C09145=1192.403,-109.333,-39.221,179.092,5.592,149.257
C09146=1192.398,-109.084,-39.231,179.093,5.592,149.257
C09147=1192.393,-108.834,-39.240,179.096,5.592,149.256
C09148=1192.388,-108.584,-39.250,179.097,5.592,149.255
C09149=1192.382,-108.334,-39.259,179.100,5.592,149.255
C09150=1192.377,-108.085,-39.269,179.102,5.592,149.254
C09151=1192.372,-107.835,-39.278,179.104,5.593,149.254
C09152=1192.367,-107.585,-39.289,179.107,5.592,149.253
C09153=1192.361,-107.335,-39.298,179.109,5.593,149.252
C09154=1192.356,-107.085,-39.308,179.111,5.593,149.252
C09155=1192.351,-106.836,-39.317,179.113,5.593,149.251
C09156=1192.345,-106.586,-39.327,179.115,5.593,149.250
C09157=1192.340,-106.337,-39.337,179.118,5.593,149.250
C09158=1192.334,-106.087,-39.346,179.119,5.593,149.249
C09159=1192.330,-105.837,-39.356,179.122,5.594,149.249
C09160=1192.324,-105.586,-39.366,179.124,5.593,149.248
C09161=1192.319,-105.337,-39.376,179.126,5.594,149.247
C09162=1192.314,-105.088,-39.385,179.128,5.594,149.247
C09163=1192.308,-104.838,-39.395,179.131,5.594,149.246
C09164=1192.303,-104.588,-39.404,179.133,5.594,149.245
C09165=1192.298,-104.338,-39.415,179.135,5.595,149.245
C09166=1192.293,-104.088,-39.424,179.137,5.595,149.244
C09167=1192.287,-103.839,-39.434,179.140,5.595,149.244
C09168=1192.282,-103.589,-39.443,179.142,5.595,149.243
C09169=1192.276,-103.339,-39.453,179.144,5.595,149.242
C09170=1192.271,-103.090,-39.463,179.147,5.596,149.242
C09171=1192.266,-102.839,-39.473,179.148,5.596,149.241
C09172=1192.261,-102.590,-39.483,179.151,5.596,149.240
C09173=1192.256,-102.340,-39.493,179.153,5.596,149.240
C09174=1192.250,-102.090,-39.502,179.155,5.597,149.239
C09175=1192.245,-101.819,-39.513,179.157,5.596,149.239
C09176=1192.239,-101.547,-39.523,179.160,5.597,149.238
C09177=1192.233,-101.276,-39.534,179.163,5.597,149.237
C09178=1192.227,-101.005,-39.545,179.165,5.597,149.236
C09179=1192.222,-100.755,-39.555,179.167,5.597,149.236
C09180=1192.217,-100.505,-39.565,179.169,5.597,149.235
C09181=1192.212,-100.255,-39.575,179.172,5.597,149.234
C09182=1192.206,-100.005,-39.584,179.173,5.597,149.234
C09183=1192.201,-99.756,-39.594,179.176,5.598,149.233
C09184=1192.196,-99.506,-39.605,179.179,5.598,149.233
C09185=1192.190,-99.256,-39.615,179.180,5.598,149.232
C09186=1192.186,-99.007,-39.624,179.183,5.599,149.231
C09187=1192.180,-98.757,-39.634,179.185,5.598,149.231
C09188=1192.175,-98.506,-39.645,179.187,5.599,149.230
C09189=1192.170,-98.257,-39.654,179.189,5.599,149.229
C09190=1192.164,-98.008,-39.664,179.191,5.599,149.229
C09191=1192.158,-97.757,-39.674,179.193,5.599,149.228
C09192=1192.153,-97.508,-39.683,179.196,5.599,149.228
C09193=1192.148,-97.258,-39.694,179.198,5.599,149.227
C09194=1192.143,-97.008,-39.704,179.200,5.600,149.226
C09195=1192.138,-96.759,-39.714,179.203,5.600,149.226
C09196=1192.133,-96.509,-39.724,179.205,5.600,149.225
C09197=1192.127,-96.259,-39.734,179.207,5.601,149.224
C09198=1192.121,-96.009,-39.744,179.209,5.600,149.224
C09199=1192.117,-95.760,-39.754,179.212,5.601,149.223
C09200=1192.112,-95.510,-39.764,179.214,5.601,149.223
C09201=1192.106,-95.260,-39.775,179.216,5.601,149.222
C09202=1192.100,-95.011,-39.785,179.218,5.601,149.221
C09203=1192.096,-94.761,-39.794,179.221,5.601,149.221
C09204=1192.090,-94.511,-39.804,179.223,5.602,149.220
C09205=1192.085,-94.261,-39.814,179.225,5.602,149.219
C09206=1192.079,-94.011,-39.825,179.228,5.602,149.219
C09207=1192.075,-93.762,-39.835,179.229,5.602,149.218
C09208=1192.069,-93.512,-39.845,179.232,5.603,149.218
C09209=1192.064,-93.262,-39.855,179.234,5.602,149.217
C09210=1192.059,-93.012,-39.866,179.236,5.603,149.216
C09211=1192.054,-92.763,-39.875,179.238,5.603,149.216
C09212=1192.048,-92.513,-39.885,179.241,5.603,149.215
C09213=1192.043,-92.263,-39.896,179.243,5.604,149.214
C09214=1192.037,-92.014,-39.906,179.245,5.604,149.214
C09215=1192.032,-91.764,-39.916,179.248,5.604,149.213
C09216=1192.028,-91.514,-39.926,179.249,5.604,149.213
C09217=1192.022,-91.265,-39.937,179.252,5.604,149.212
C09218=1192.016,-91.015,-39.947,179.254,5.604,149.211
C09219=1192.011,-90.765,-39.957,179.256,5.605,149.211
C09220=1192.006,-90.515,-39.968,179.258,5.604,149.210
C09221=1192.000,-90.266,-39.978,179.261,5.605,149.209
C09222=1191.996,-90.016,-39.988,179.263,5.606,149.209
C09223=1191.990,-89.766,-39.998,179.265,5.605,149.208
C09224=1191.985,-89.517,-40.008,179.268,5.606,149.207
C09225=1191.980,-89.266,-40.019,179.270,5.606,149.207
C09226=1191.974,-89.017,-40.029,179.272,5.606,149.206
C09227=1191.969,-88.767,-40.039,179.274,5.606,149.205
C09228=1191.964,-88.517,-40.049,179.277,5.606,149.205
C09229=1191.959,-88.268,-40.059,179.279,5.607,149.204
C09230=1191.954,-88.018,-40.070,179.281,5.606,149.203
C09231=1191.948,-87.768,-40.080,179.284,5.607,149.203
C09232=1191.943,-87.519,-40.090,179.286,5.607,149.202
C09233=1191.938,-87.268,-40.101,179.288,5.607,149.202
C09234=1191.932,-87.019,-40.111,179.290,5.607,149.201
C09235=1191.927,-86.769,-40.122,179.293,5.608,149.200
C09236=1191.921,-86.519,-40.132,179.295,5.608,149.200
C09237=1191.917,-86.270,-40.142,179.297,5.608,149.199
C09238=1191.912,-86.020,-40.153,179.300,5.608,149.198
C09239=1191.906,-85.771,-40.163,179.302,5.608,149.198
C09240=1191.901,-85.520,-40.174,179.304,5.609,149.197
C09241=1191.896,-85.271,-40.184,179.307,5.609,149.197
C09242=1191.891,-85.021,-40.194,179.309,5.609,149.196
C09243=1191.885,-84.771,-40.205,179.311,5.609,149.195
C09244=1191.880,-84.522,-40.216,179.313,5.609,149.195
C09245=1191.875,-84.272,-40.226,179.316,5.610,149.194
C09246=1191.869,-84.022,-40.236,179.318,5.609,149.193
C09247=1191.864,-83.772,-40.247,179.320,5.610,149.193
C09248=1191.859,-83.523,-40.257,179.322,5.611,149.192
C09249=1191.854,-83.273,-40.268,179.325,5.610,149.191
C09250=1191.848,-83.023,-40.279,179.327,5.611,149.191
C09251=1191.843,-82.773,-40.289,179.329,5.611,149.190
C09252=1191.838,-82.524,-40.299,179.331,5.611,149.189
C09253=1191.832,-82.274,-40.310,179.334,5.611,149.189
C09254=1191.827,-82.024,-40.321,179.336,5.611,149.188
C09255=1191.822,-81.775,-40.331,179.338,5.612,149.188
C09256=1191.817,-81.525,-40.342,179.341,5.611,149.187
C09257=1191.811,-81.275,-40.352,179.343,5.612,149.186
C09258=1191.806,-81.025,-40.363,179.345,5.613,149.186
C09259=1191.801,-80.776,-40.373,179.347,5.612,149.185
C09260=1191.796,-80.526,-40.384,179.350,5.613,149.184
C09261=1191.790,-80.276,-40.394,179.352,5.613,149.184
C09262=1191.786,-80.027,-40.405,179.354,5.613,149.183
C09263=1191.780,-79.777,-40.416,179.357,5.614,149.182
C09264=1191.775,-79.527,-40.426,179.359,5.614,149.182
C09265=1191.770,-79.278,-40.437,179.361,5.614,149.181
C09266=1191.765,-79.028,-40.448,179.363,5.614,149.180
C09267=1191.759,-78.778,-40.458,179.366,5.614,149.180
C09268=1191.754,-78.528,-40.469,179.368,5.615,149.179
C09269=1191.749,-78.279,-40.479,179.370,5.614,149.179
C09270=1191.744,-78.029,-40.490,179.373,5.615,149.178
C09271=1191.739,-77.780,-40.501,179.375,5.615,149.177
C09272=1191.734,-77.529,-40.512,179.377,5.615,149.177
C09273=1191.728,-77.280,-40.522,179.380,5.616,149.176
C09274=1191.723,-77.030,-40.533,179.382,5.616,149.175
C09275=1191.717,-76.780,-40.544,179.384,5.616,149.175
C09276=1191.712,-76.530,-40.554,179.386,5.616,149.174
C09277=1191.707,-76.281,-40.565,179.389,5.617,149.174
C09278=1191.702,-76.031,-40.576,179.391,5.617,149.173
C09279=1191.696,-75.760,-40.588,179.393,5.617,149.172
C09280=1191.691,-75.490,-40.599,179.396,5.617,149.171
C09281=1191.685,-75.218,-40.611,179.399,5.617,149.171
C09282=1191.679,-74.947,-40.623,179.401,5.618,149.170
C09283=1191.673,-74.698,-40.633,179.403,5.618,149.169
C09284=1191.669,-74.448,-40.645,179.406,5.618,149.169
C09285=1191.663,-74.199,-40.655,179.408,5.619,149.168
C09286=1191.658,-73.949,-40.666,179.410,5.618,149.167
C09287=1191.653,-73.700,-40.676,179.412,5.619,149.167
C09288=1191.647,-73.450,-40.688,179.415,5.619,149.166
C09289=1191.642,-73.200,-40.699,179.417,5.619,149.166
C09290=1191.637,-72.950,-40.710,179.420,5.620,149.165
C09291=1191.632,-72.700,-40.720,179.422,5.620,149.164
C09292=1191.627,-72.451,-40.731,179.424,5.620,149.164
C09293=1191.621,-72.201,-40.743,179.427,5.620,149.163
C09294=1191.616,-71.952,-40.753,179.428,5.620,149.162
C09295=1191.611,-71.702,-40.764,179.431,5.621,149.162
C09296=1191.606,-71.452,-40.775,179.433,5.621,149.161
C09297=1191.600,-71.202,-40.786,179.436,5.621,149.160
C09298=1191.595,-70.952,-40.797,179.438,5.622,149.160
C09299=1191.589,-70.703,-40.808,179.440,5.621,149.159
C09300=1191.585,-70.453,-40.819,179.443,5.622,149.158
C09301=1191.580,-70.203,-40.829,179.445,5.623,149.158
C09302=1191.574,-69.954,-40.841,179.447,5.622,149.157
C09303=1191.569,-69.704,-40.852,179.450,5.623,149.157
C09304=1191.564,-69.454,-40.863,179.452,5.622,149.156
C09305=1191.559,-69.205,-40.874,179.454,5.623,149.155
C09306=1191.553,-68.954,-40.885,179.457,5.624,149.155
C09307=1191.548,-68.706,-40.896,179.459,5.623,149.154
C09308=1191.543,-68.456,-40.907,179.461,5.624,149.153
C09309=1191.538,-68.206,-40.918,179.464,5.624,149.153
C09310=1191.532,-67.956,-40.929,179.466,5.624,149.152
C09311=1191.527,-67.706,-40.940,179.468,5.624,149.151
C09312=1191.522,-67.457,-40.951,179.471,5.625,149.151
C09313=1191.516,-67.207,-40.963,179.473,5.625,149.150
C09314=1191.511,-66.957,-40.973,179.475,5.625,149.149
C09315=1191.507,-66.707,-40.984,179.478,5.626,149.149
C09316=1191.501,-66.458,-40.996,179.480,5.626,149.148
C09317=1191.496,-66.208,-41.007,179.482,5.626,149.148
C09318=1191.491,-65.958,-41.018,179.484,5.626,149.147
C09319=1191.486,-65.709,-41.029,179.487,5.626,149.146
C09320=1191.480,-65.459,-41.040,179.489,5.627,149.146
C09321=1191.475,-65.209,-41.051,179.491,5.627,149.145
C09322=1191.470,-64.960,-41.063,179.494,5.627,149.144
C09323=1191.464,-64.710,-41.074,179.496,5.628,149.144
C09324=1191.459,-64.460,-41.085,179.498,5.628,149.143
C09325=1191.454,-64.210,-41.097,179.501,5.628,149.142
C09326=1191.449,-63.961,-41.107,179.504,5.628,149.142
C09327=1191.444,-63.712,-41.119,179.505,5.628,149.141
C09328=1191.438,-63.461,-41.130,179.508,5.629,149.140
C09329=1191.433,-63.212,-41.141,179.510,5.629,149.140
C09330=1191.428,-62.963,-41.152,179.513,5.629,149.139
C09331=1191.423,-62.713,-41.164,179.515,5.630,149.139
C09332=1191.418,-62.462,-41.175,179.517,5.630,149.138
C09333=1191.412,-62.213,-41.186,179.519,5.630,149.137
C09334=1191.407,-61.964,-41.197,179.522,5.630,149.136
C09335=1191.402,-61.714,-41.209,179.524,5.631,149.136
C09336=1191.397,-61.464,-41.221,179.526,5.631,149.135
C09337=1191.391,-61.214,-41.231,179.529,5.631,149.135
C09338=1191.386,-60.964,-41.243,179.532,5.632,149.134
C09339=1191.381,-60.715,-41.254,179.533,5.632,149.133
C09340=1191.377,-60.465,-41.265,179.536,5.632,149.133
C09341=1191.371,-60.216,-41.277,179.539,5.632,149.132
C09342=1191.366,-59.966,-41.288,179.540,5.632,149.131
C09343=1191.360,-59.716,-41.299,179.543,5.633,149.131
C09344=1191.355,-59.466,-41.311,179.546,5.633,149.130
C09345=1191.350,-59.216,-41.322,179.548,5.633,149.129
C09346=1191.345,-58.967,-41.333,179.550,5.634,149.129
C09347=1191.339,-58.717,-41.345,179.553,5.634,149.128
C09348=1191.335,-58.468,-41.357,179.555,5.634,149.127
C09349=1191.329,-58.218,-41.368,179.557,5.634,149.127
C09350=1191.324,-57.969,-41.379,179.559,5.635,149.126
C09351=1191.319,-57.719,-41.391,179.562,5.635,149.126
C09352=1191.314,-57.469,-41.402,179.564,5.635,149.125
C09353=1191.309,-57.220,-41.414,179.567,5.636,149.124
C09354=1191.304,-56.970,-41.426,179.568,5.636,149.124
C09355=1191.299,-56.720,-41.436,179.571,5.636,149.123
C09356=1191.293,-56.470,-41.448,179.574,5.636,149.122
C09357=1191.288,-56.221,-41.459,179.576,5.637,149.122
C09358=1191.282,-55.971,-41.471,179.578,5.637,149.121
C09359=1191.277,-55.721,-41.483,179.581,5.637,149.120
C09360=1191.272,-55.471,-41.494,179.583,5.638,149.120
C09361=1191.266,-55.222,-41.506,179.585,5.637,149.119
C09362=1191.262,-54.972,-41.517,179.588,5.638,149.119
C09363=1191.256,-54.722,-41.529,179.590,5.639,149.118
C09364=1191.252,-54.473,-41.540,179.592,5.638,149.117
C09365=1191.246,-54.223,-41.552,179.595,5.639,149.116
C09366=1191.241,-53.973,-41.563,179.597,5.640,149.116
C09367=1191.236,-53.723,-41.575,179.599,5.639,149.115
C09368=1191.231,-53.475,-41.587,179.602,5.640,149.115
C09369=1191.226,-53.225,-41.599,179.605,5.640,149.114
C09370=1191.220,-52.975,-41.611,179.607,5.641,149.113
C09371=1191.215,-52.725,-41.622,179.609,5.641,149.113
C09372=1191.210,-52.476,-41.634,179.612,5.641,149.112
C09373=1191.205,-52.226,-41.645,179.614,5.641,149.111
C09374=1191.200,-51.976,-41.657,179.616,5.641,149.111
C09375=1191.194,-51.726,-41.669,179.619,5.642,149.110
C09376=1191.189,-51.477,-41.680,179.621,5.642,149.109
C09377=1191.184,-51.227,-41.692,179.623,5.642,149.109
C09378=1191.179,-50.978,-41.703,179.625,5.643,149.108
C09379=1191.174,-50.728,-41.715,179.628,5.643,149.107
C09380=1191.168,-50.478,-41.727,179.631,5.644,149.107
C09381=1191.164,-50.229,-41.739,179.633,5.643,149.106
C09382=1191.158,-49.979,-41.751,179.635,5.644,149.106
C09383=1191.152,-49.709,-41.763,179.638,5.645,149.105
C09384=1191.147,-49.439,-41.776,179.640,5.645,149.104
C09385=1191.142,-49.168,-41.788,179.643,5.645,149.104
C09386=1191.136,-48.898,-41.801,179.645,5.645,149.103
C09387=1191.131,-48.649,-41.814,179.648,5.645,149.102
C09388=1191.125,-48.399,-41.825,179.650,5.646,149.101
C09389=1191.120,-48.149,-41.837,179.653,5.646,149.101
C09390=1191.115,-47.899,-41.849,179.655,5.646,149.100
C09391=1191.110,-47.649,-41.861,179.657,5.647,149.100
C09392=1191.105,-47.400,-41.873,179.660,5.647,149.099
C09393=1191.100,-47.150,-41.884,179.662,5.647,149.098
C09394=1191.094,-46.900,-41.896,179.664,5.648,149.098
C09395=1191.089,-46.650,-41.908,179.667,5.648,149.097
C09396=1191.084,-46.401,-41.920,179.670,5.649,149.096
C09397=1191.079,-46.152,-41.932,179.672,5.648,149.096
C09398=1191.074,-45.902,-41.944,179.674,5.649,149.095
C09399=1191.068,-45.652,-41.956,179.677,5.650,149.094
C09400=1191.064,-45.403,-41.968,179.679,5.649,149.094
C09401=1191.058,-45.153,-41.980,179.681,5.650,149.093
C09402=1191.052,-44.904,-41.991,179.684,5.650,149.092
C09403=1191.047,-44.654,-42.004,179.686,5.651,149.092
C09404=1191.043,-44.405,-42.015,179.688,5.651,149.091
C09405=1191.037,-44.155,-42.027,179.691,5.651,149.090
C09406=1191.032,-43.905,-42.039,179.694,5.651,149.090
C09407=1191.027,-43.655,-42.052,179.696,5.652,149.089
C09408=1191.022,-43.406,-42.063,179.698,5.652,149.089
C09409=1191.017,-43.156,-42.075,179.700,5.652,149.088
C09410=1191.011,-42.906,-42.087,179.703,5.653,149.087
C09411=1191.006,-42.657,-42.099,179.705,5.654,149.087
C09412=1191.001,-42.407,-42.112,179.707,5.653,149.086
C09413=1190.995,-42.157,-42.124,179.710,5.654,149.085
C09414=1190.991,-41.908,-42.135,179.713,5.654,149.085
C09415=1190.986,-41.658,-42.148,179.714,5.654,149.084
C09416=1190.981,-41.408,-42.160,179.717,5.655,149.083
C09417=1190.976,-41.158,-42.172,179.720,5.655,149.083
C09418=1190.970,-40.908,-42.184,179.722,5.656,149.082
C09419=1190.965,-40.659,-42.196,179.724,5.655,149.081
C09420=1190.960,-40.410,-42.208,179.727,5.656,149.081
C09421=1190.955,-40.160,-42.220,179.729,5.656,149.080
C09422=1190.950,-39.910,-42.233,179.732,5.657,149.079
C09423=1190.944,-39.660,-42.245,179.734,5.657,149.079
C09424=1190.939,-39.411,-42.257,179.736,5.657,149.078
C09425=1190.934,-39.161,-42.269,179.739,5.658,149.078
C09426=1190.929,-38.912,-42.282,179.741,5.658,149.077
C09427=1190.923,-38.662,-42.294,179.744,5.658,149.076
C09428=1190.919,-38.413,-42.306,179.746,5.659,149.076
C09429=1190.913,-38.163,-42.317,179.748,5.659,149.075
C09430=1190.908,-37.914,-42.330,179.751,5.660,149.074
C09431=1190.903,-37.664,-42.342,179.753,5.659,149.074
C09432=1190.898,-37.414,-42.354,179.756,5.660,149.073
C09433=1190.893,-37.164,-42.367,179.758,5.661,149.072
C09434=1190.888,-36.914,-42.379,179.761,5.661,149.072
C09435=1190.882,-36.664,-42.391,179.763,5.661,149.071
C09436=1190.877,-36.415,-42.404,179.765,5.661,149.070
C09437=1190.872,-36.165,-42.416,179.768,5.662,149.070
C09438=1190.867,-35.916,-42.428,179.770,5.662,149.069
C09439=1190.862,-35.667,-42.441,179.773,5.663,149.068
C09440=1190.856,-35.417,-42.453,179.775,5.662,149.068
C09441=1190.851,-35.167,-42.465,179.777,5.663,149.067
C09442=1190.846,-34.917,-42.477,179.780,5.664,149.067
C09443=1190.841,-34.667,-42.490,179.782,5.664,149.066
C09444=1190.836,-34.418,-42.503,179.785,5.664,149.065
C09445=1190.830,-34.168,-42.515,179.787,5.664,149.064
C09446=1190.825,-33.919,-42.527,179.789,5.665,149.064
C09447=1190.820,-33.669,-42.539,179.792,5.666,149.063
C09448=1190.815,-33.419,-42.552,179.795,5.666,149.063
C09449=1190.810,-33.170,-42.564,179.797,5.666,149.062
C09450=1190.805,-32.920,-42.577,179.799,5.667,149.061
C09451=1190.800,-32.670,-42.589,179.802,5.667,149.061
C09452=1190.795,-32.421,-42.602,179.804,5.667,149.060
C09453=1190.789,-32.171,-42.614,179.806,5.667,149.059
C09454=1190.784,-31.922,-42.626,179.809,5.668,149.059
C09455=1190.779,-31.672,-42.639,179.811,5.668,149.058
C09456=1190.773,-31.422,-42.651,179.814,5.669,149.057
C09457=1190.769,-31.172,-42.664,179.817,5.669,149.057
C09458=1190.764,-30.923,-42.676,179.819,5.669,149.056
C09459=1190.759,-30.674,-42.689,179.821,5.670,149.056
C09460=1190.753,-30.424,-42.701,179.823,5.670,149.055
C09461=1190.748,-30.174,-42.714,179.826,5.671,149.054
C09462=1190.744,-29.924,-42.726,179.829,5.671,149.053
C09463=1190.739,-29.675,-42.739,179.830,5.671,149.053
C09464=1190.732,-29.425,-42.752,179.833,5.672,149.052
C09465=1190.727,-29.176,-42.764,179.836,5.672,149.052
C09466=1190.722,-28.926,-42.777,179.838,5.673,149.051
C09467=1190.718,-28.676,-42.790,179.840,5.673,149.050
C09468=1190.712,-28.427,-42.802,179.843,5.673,149.050
C09469=1190.707,-28.177,-42.814,179.845,5.674,149.049
C09470=1190.702,-27.928,-42.827,179.848,5.674,149.048
C09471=1190.697,-27.678,-42.839,179.851,5.674,149.048
C09472=1190.692,-27.428,-42.852,179.853,5.675,149.047
C09473=1190.686,-27.179,-42.866,179.855,5.675,149.046
C09474=1190.681,-26.929,-42.878,179.857,5.675,149.046
C09475=1190.676,-26.679,-42.890,179.860,5.676,149.045
C09476=1190.671,-26.429,-42.903,179.862,5.677,149.045
C09477=1190.666,-26.180,-42.916,179.865,5.677,149.044
C09478=1190.661,-25.931,-42.928,179.867,5.677,149.043
C09479=1190.655,-25.681,-42.941,179.870,5.677,149.043
C09480=1190.651,-25.431,-42.954,179.872,5.678,149.042
C09481=1190.646,-25.182,-42.967,179.875,5.679,149.041
C09482=1190.640,-24.933,-42.980,179.877,5.679,149.041
C09483=1190.636,-24.682,-42.992,179.879,5.679,149.040
C09484=1190.630,-24.433,-43.004,179.882,5.679,149.039
C09485=1190.625,-24.183,-43.018,179.884,5.680,149.039
C09486=1190.619,-23.934,-43.030,179.887,5.680,149.038
C09487=1190.614,-23.664,-43.044,179.889,5.681,149.037
C09488=1190.609,-23.394,-43.058,179.892,5.681,149.037
C09489=1190.603,-23.125,-43.072,179.895,5.682,149.036
C09490=1190.597,-22.855,-43.086,179.897,5.682,149.035
C09491=1190.592,-22.605,-43.098,179.900,5.683,149.035
C09492=1190.588,-22.355,-43.111,179.902,5.682,149.034
C09493=1190.582,-22.106,-43.125,179.904,5.683,149.033
C09494=1190.577,-21.857,-43.137,179.907,5.684,149.033
C09495=1190.572,-21.606,-43.150,179.910,5.684,149.032
C09496=1190.567,-21.357,-43.163,179.912,5.685,149.031
C09497=1190.561,-21.108,-43.176,179.914,5.685,149.031
C09498=1190.557,-20.858,-43.189,179.917,5.685,149.030
C09499=1190.552,-20.608,-43.201,179.919,5.686,149.030
C09500=1190.546,-20.359,-43.215,179.922,5.686,149.029
C09501=1190.541,-20.109,-43.228,179.925,5.686,149.028
C09502=1190.536,-19.860,-43.241,179.927,5.687,149.028
C09503=1190.531,-19.611,-43.254,179.929,5.688,149.027
C09504=1190.526,-19.360,-43.267,179.931,5.687,149.026
C09505=1190.521,-19.111,-43.280,179.934,5.688,149.026
C09506=1190.516,-18.862,-43.292,179.936,5.689,149.025
C09507=1190.511,-18.611,-43.306,179.939,5.689,149.024
C09508=1190.505,-18.362,-43.318,179.942,5.690,149.024
C09509=1190.500,-18.113,-43.331,179.944,5.690,149.023
C09510=1190.495,-17.862,-43.345,179.946,5.690,149.022
C09511=1190.490,-17.613,-43.357,179.948,5.691,149.022
C09512=1190.484,-17.364,-43.371,179.951,5.691,149.021
C09513=1190.480,-17.114,-43.384,179.954,5.692,149.020
C09514=1190.475,-16.865,-43.397,179.956,5.692,149.020
C09515=1190.469,-16.614,-43.410,179.959,5.693,149.019
C09516=1190.464,-16.365,-43.423,179.961,5.693,149.019
C09517=1190.459,-16.116,-43.435,179.963,5.693,149.018
C09518=1190.454,-15.866,-43.450,179.966,5.694,149.017
C09519=1190.449,-15.617,-43.462,179.968,5.694,149.017
C09520=1190.444,-15.366,-43.476,179.971,5.695,149.016
C09521=1190.439,-15.117,-43.489,179.974,5.695,149.015
C09522=1190.434,-14.868,-43.501,179.976,5.696,149.015
C09523=1190.429,-14.618,-43.515,179.979,5.696,149.014
C09524=1190.424,-14.369,-43.528,179.980,5.696,149.014
C09525=1190.418,-14.118,-43.542,179.983,5.697,149.013
C09526=1190.413,-13.869,-43.554,179.986,5.697,149.012
C09527=1190.408,-13.619,-43.568,179.988,5.698,149.011
C09528=1190.403,-13.370,-43.581,179.991,5.699,149.011
C09529=1190.397,-13.120,-43.594,179.993,5.699,149.010
C09530=1190.393,-12.870,-43.607,179.996,5.699,149.010
C09531=1190.388,-12.622,-43.621,179.998,5.699,149.009
C09532=1190.383,-12.371,-43.634,-180.000,5.700,149.008
C09533=1190.377,-12.122,-43.647,-179.997,5.700,149.008
C09534=1190.373,-11.872,-43.661,-179.995,5.701,149.007
C09535=1190.367,-11.623,-43.674,-179.992,5.701,149.006
C09536=1190.362,-11.373,-43.687,-179.989,5.702,149.006
C09537=1190.357,-11.124,-43.700,-179.987,5.703,149.005
C09538=1190.352,-10.874,-43.714,-179.984,5.703,149.005
C09539=1190.347,-10.624,-43.727,-179.982,5.703,149.004
C09540=1190.342,-10.375,-43.741,-179.980,5.703,149.003
C09541=1190.337,-10.125,-43.753,-179.978,5.704,149.003
C09542=1190.331,-9.876,-43.767,-179.975,5.705,149.002
C09543=1190.327,-9.626,-43.780,-179.972,5.705,149.001
C09544=1190.321,-9.377,-43.794,-179.970,5.706,149.001
C09545=1190.316,-9.127,-43.808,-179.967,5.706,149.000
C09546=1190.311,-8.878,-43.820,-179.965,5.707,148.999
C09547=1190.306,-8.628,-43.835,-179.962,5.707,148.999
C09548=1190.301,-8.378,-43.848,-179.960,5.707,148.998
C09549=1190.295,-8.128,-43.861,-179.958,5.708,148.998
C09550=1190.291,-7.879,-43.875,-179.955,5.708,148.997
C09551=1190.285,-7.629,-43.888,-179.953,5.709,148.996
C09552=1190.281,-7.380,-43.901,-179.950,5.709,148.996
C09553=1190.275,-7.130,-43.915,-179.947,5.710,148.995
C09554=1190.270,-6.880,-43.929,-179.945,5.711,148.994
C09555=1190.265,-6.631,-43.942,-179.942,5.711,148.994
C09556=1190.260,-6.381,-43.956,-179.940,5.712,148.993
C09557=1190.255,-6.132,-43.968,-179.938,5.711,148.992
C09558=1190.250,-5.882,-43.983,-179.936,5.712,148.992
C09559=1190.244,-5.633,-43.996,-179.933,5.713,148.991
C09560=1190.240,-5.383,-44.010,-179.930,5.713,148.990
C09561=1190.235,-5.133,-44.023,-179.928,5.714,148.990
C09562=1190.229,-4.884,-44.037,-179.925,5.714,148.989
C09563=1190.225,-4.634,-44.050,-179.923,5.715,148.989
C09564=1190.219,-4.385,-44.064,-179.920,5.715,148.988
C09565=1190.214,-4.135,-44.077,-179.917,5.716,148.987
C09566=1190.209,-3.886,-44.091,-179.915,5.717,148.987
C09567=1190.204,-3.636,-44.105,-179.913,5.717,148.986
C09568=1190.199,-3.386,-44.119,-179.911,5.717,148.985
C09569=1190.194,-3.137,-44.132,-179.908,5.717,148.985
C09570=1190.189,-2.887,-44.145,-179.905,5.718,148.984
C09571=1190.183,-2.638,-44.159,-179.903,5.719,148.984
C09572=1190.179,-2.388,-44.173,-179.900,5.719,148.983
C09573=1190.174,-2.138,-44.187,-179.898,5.720,148.982
C09574=1190.168,-1.889,-44.201,-179.895,5.720,148.981
C09575=1190.164,-1.640,-44.214,-179.893,5.721,148.981
C09576=1190.158,-1.390,-44.227,-179.890,5.721,148.980
C09577=1190.153,-1.140,-44.242,-179.888,5.722,148.980
C09578=1190.148,-0.891,-44.256,-179.885,5.722,148.979
C09579=1190.143,-0.641,-44.269,-179.883,5.723,148.978
C09580=1190.138,-0.392,-44.283,-179.881,5.723,148.978
C09581=1190.133,-0.142,-44.297,-179.878,5.723,148.977
C09582=1190.127,0.108,-44.310,-179.875,5.724,148.976
C09583=1190.123,0.357,-44.324,-179.873,5.725,148.976
C09584=1190.118,0.606,-44.338,-179.871,5.725,148.975
C09585=1190.112,0.856,-44.351,-179.868,5.726,148.975
C09586=1190.107,1.106,-44.366,-179.865,5.726,148.974
C09587=1190.102,1.355,-44.380,-179.863,5.727,148.973
C09588=1190.098,1.605,-44.393,-179.860,5.727,148.973
C09589=1190.092,1.855,-44.407,-179.858,5.728,148.972
C09590=1190.087,2.104,-44.421,-179.855,5.728,148.971
C09591=1190.081,2.373,-44.436,-179.852,5.729,148.971
C09592=1190.076,2.643,-44.451,-179.850,5.729,148.970
C09593=1190.071,2.912,-44.467,-179.847,5.730,148.969
C09594=1190.065,3.181,-44.482,-179.845,5.730,148.969
C09595=1190.060,3.430,-44.495,-179.842,5.731,148.968
C09596=1190.055,3.680,-44.508,-179.840,5.732,148.967
C09597=1190.050,3.930,-44.523,-179.837,5.732,148.967
C09598=1190.045,4.179,-44.537,-179.834,5.733,148.966
C09599=1190.040,4.428,-44.551,-179.832,5.734,148.966
C09600=1190.035,4.678,-44.565,-179.830,5.734,148.965
C09601=1190.030,4.928,-44.579,-179.827,5.734,148.964
C09602=1190.024,5.177,-44.593,-179.824,5.735,148.964
C09603=1190.020,5.427,-44.606,-179.822,5.736,148.963
C09604=1190.015,5.677,-44.621,-179.819,5.736,148.962
C09605=1190.009,5.926,-44.634,-179.817,5.737,148.962
C09606=1190.004,6.175,-44.649,-179.814,5.737,148.961
C09607=1189.999,6.425,-44.663,-179.812,5.738,148.961
C09608=1189.994,6.675,-44.677,-179.809,5.739,148.960
C09609=1189.989,6.924,-44.691,-179.807,5.739,148.959
C09610=1189.984,7.173,-44.706,-179.804,5.740,148.959
C09611=1189.979,7.423,-44.720,-179.802,5.740,148.958
C09612=1189.974,7.673,-44.734,-179.800,5.740,148.957
C09613=1189.969,7.922,-44.748,-179.797,5.741,148.957
C09614=1189.964,8.171,-44.762,-179.794,5.741,148.956
C09615=1189.959,8.421,-44.776,-179.792,5.742,148.956
C09616=1189.954,8.671,-44.789,-179.790,5.742,148.955
C09617=1189.949,8.920,-44.803,-179.787,5.743,148.954
C09618=1189.944,9.170,-44.818,-179.784,5.743,148.954
C09619=1189.939,9.420,-44.832,-179.782,5.744,148.953
C09620=1189.934,9.669,-44.846,-179.780,5.745,148.952
C09621=1189.929,9.919,-44.861,-179.777,5.745,148.952
C09622=1189.923,10.168,-44.875,-179.774,5.746,148.951
C09623=1189.919,10.417,-44.889,-179.772,5.747,148.951
C09624=1189.914,10.667,-44.904,-179.769,5.747,148.950
C09625=1189.909,10.917,-44.918,-179.767,5.748,148.949
C09626=1189.904,11.166,-44.932,-179.764,5.748,148.948
C09627=1189.898,11.415,-44.946,-179.762,5.749,148.948
C09628=1189.893,11.665,-44.960,-179.759,5.749,148.947
C09629=1189.888,11.915,-44.975,-179.757,5.750,148.947
C09630=1189.883,12.164,-44.989,-179.755,5.751,148.946
C09631=1189.878,12.414,-45.003,-179.752,5.751,148.946
C09632=1189.873,12.664,-45.018,-179.749,5.752,148.945
C09633=1189.867,12.913,-45.032,-179.747,5.752,148.944
C09634=1189.862,13.162,-45.047,-179.744,5.753,148.944
C09635=1189.857,13.412,-45.061,-179.742,5.754,148.943
C09636=1189.852,13.662,-45.076,-179.739,5.754,148.942
C09637=1189.848,13.911,-45.090,-179.736,5.755,148.942
C09638=1189.843,14.161,-45.104,-179.734,5.755,148.941
C09639=1189.837,14.410,-45.118,-179.732,5.756,148.941
C09640=1189.832,14.659,-45.133,-179.729,5.756,148.940
C09641=1189.827,14.909,-45.147,-179.726,5.757,148.939
C09642=1189.822,15.159,-45.162,-179.724,5.758,148.939
C09643=1189.817,15.408,-45.176,-179.722,5.758,148.938
C09644=1189.812,15.658,-45.191,-179.719,5.759,148.937
C09645=1189.807,15.908,-45.206,-179.716,5.759,148.937
C09646=1189.802,16.157,-45.220,-179.714,5.760,148.936
C09647=1189.797,16.407,-45.234,-179.711,5.761,148.936
C09648=1189.792,16.656,-45.248,-179.709,5.761,148.935
C09649=1189.787,16.905,-45.263,-179.707,5.762,148.934
C09650=1189.782,17.155,-45.277,-179.704,5.763,148.934
C09651=1189.776,17.405,-45.292,-179.701,5.763,148.933
C09652=1189.771,17.654,-45.307,-179.699,5.763,148.932
C09653=1189.767,17.904,-45.322,-179.696,5.764,148.932
C09654=1189.762,18.153,-45.336,-179.694,5.765,148.931
C09655=1189.757,18.403,-45.350,-179.691,5.765,148.930
C09656=1189.752,18.652,-45.365,-179.689,5.766,148.930
C09657=1189.747,18.902,-45.380,-179.686,5.767,148.929
C09658=1189.742,19.152,-45.394,-179.684,5.767,148.929
C09659=1189.737,19.401,-45.409,-179.681,5.768,148.928
C09660=1189.731,19.650,-45.423,-179.678,5.768,148.927
C09661=1189.726,19.900,-45.438,-179.676,5.769,148.927
C09662=1189.721,20.149,-45.453,-179.674,5.770,148.926
C09663=1189.716,20.399,-45.467,-179.671,5.770,148.926
C09664=1189.711,20.648,-45.482,-179.669,5.771,148.925
C09665=1189.706,20.898,-45.497,-179.666,5.772,148.924
C09666=1189.701,21.148,-45.512,-179.663,5.773,148.924
C09667=1189.696,21.397,-45.527,-179.660,5.773,148.923
C09668=1189.691,21.646,-45.541,-179.658,5.774,148.923
C09669=1189.686,21.896,-45.555,-179.655,5.775,148.922
C09670=1189.681,22.145,-45.571,-179.653,5.775,148.921
C09671=1189.676,22.395,-45.585,-179.651,5.776,148.921
C09672=1189.671,22.644,-45.600,-179.648,5.776,148.920
C09673=1189.666,22.894,-45.615,-179.645,5.777,148.919
C09674=1189.661,23.143,-45.630,-179.643,5.777,148.919
C09675=1189.656,23.393,-45.644,-179.641,5.778,148.918
C09676=1189.651,23.642,-45.659,-179.638,5.779,148.918
C09677=1189.646,23.892,-45.674,-179.635,5.779,148.917
C09678=1189.641,24.141,-45.689,-179.633,5.780,148.916
C09679=1189.636,24.391,-45.703,-179.630,5.781,148.916
C09680=1189.631,24.640,-45.719,-179.628,5.781,148.915
C09681=1189.626,24.890,-45.733,-179.625,5.782,148.914
C09682=1189.621,25.139,-45.748,-179.623,5.783,148.914
C09683=1189.615,25.389,-45.763,-179.620,5.783,148.913
C09684=1189.611,25.638,-45.778,-179.618,5.784,148.913
C09685=1189.606,25.888,-45.792,-179.615,5.784,148.912
C09686=1189.600,26.137,-45.808,-179.612,5.786,148.911
C09687=1189.595,26.387,-45.822,-179.610,5.786,148.911
C09688=1189.590,26.637,-45.838,-179.607,5.787,148.910
C09689=1189.585,26.886,-45.853,-179.605,5.788,148.910
C09690=1189.581,27.136,-45.867,-179.602,5.788,148.909
C09691=1189.576,27.385,-45.883,-179.600,5.789,148.908
C09692=1189.571,27.635,-45.897,-179.597,5.790,148.908
C09693=1189.565,27.885,-45.913,-179.595,5.790,148.907
C09694=1189.561,28.134,-45.928,-179.592,5.791,148.906
C09695=1189.555,28.402,-45.943,-179.589,5.791,148.906
C09696=1189.550,28.672,-45.960,-179.586,5.792,148.905
C09697=1189.545,28.940,-45.976,-179.584,5.793,148.904
C09698=1189.539,29.209,-45.992,-179.581,5.793,148.904
C09699=1189.534,29.458,-46.007,-179.579,5.794,148.903
C09700=1189.529,29.708,-46.022,-179.576,5.795,148.903
C09701=1189.524,29.957,-46.037,-179.574,5.795,148.902
C09702=1189.519,30.206,-46.053,-179.571,5.796,148.902
C09703=1189.514,30.456,-46.067,-179.569,5.797,148.901
C09704=1189.508,30.706,-46.083,-179.565,5.798,148.900
C09705=1189.504,30.955,-46.098,-179.563,5.798,148.899
C09706=1189.499,31.205,-46.114,-179.561,5.799,148.899
C09707=1189.494,31.454,-46.128,-179.558,5.800,148.898
C09708=1189.488,31.704,-46.144,-179.555,5.800,148.898
C09709=1189.484,31.953,-46.159,-179.553,5.801,148.897
C09710=1189.478,32.202,-46.174,-179.551,5.802,148.897
C09711=1189.473,32.452,-46.188,-179.548,5.802,148.896
C09712=1189.469,32.702,-46.204,-179.546,5.803,148.895
C09713=1189.464,32.951,-46.219,-179.543,5.804,148.895
C09714=1189.459,33.201,-46.235,-179.541,5.804,148.894
C09715=1189.454,33.450,-46.250,-179.537,5.805,148.893
C09716=1189.448,33.700,-46.265,-179.535,5.806,148.893
C09717=1189.443,33.949,-46.280,-179.532,5.807,148.892
C09718=1189.439,34.199,-46.296,-179.530,5.807,148.892
C09719=1189.433,34.448,-46.311,-179.528,5.808,148.891
C09720=1189.429,34.697,-46.326,-179.525,5.809,148.890
C09721=1189.423,34.947,-46.342,-179.522,5.809,148.890
C09722=1189.419,35.196,-46.357,-179.520,5.810,148.889
C09723=1189.413,35.446,-46.372,-179.518,5.811,148.889
C09724=1189.408,35.696,-46.388,-179.514,5.812,148.888
C09725=1189.404,35.945,-46.403,-179.512,5.813,148.888
C09726=1189.398,36.195,-46.418,-179.510,5.813,148.887
C09727=1189.394,36.444,-46.433,-179.507,5.814,148.886
C09728=1189.388,36.693,-46.449,-179.505,5.815,148.886
C09729=1189.383,36.943,-46.465,-179.502,5.815,148.885
C09730=1189.379,37.192,-46.480,-179.500,5.816,148.884
C09731=1189.373,37.442,-46.495,-179.497,5.816,148.884
C09732=1189.368,37.691,-46.511,-179.494,5.818,148.883
C09733=1189.364,37.941,-46.526,-179.491,5.818,148.883
C09734=1189.359,38.190,-46.542,-179.489,5.819,148.882
C09735=1189.353,38.440,-46.558,-179.487,5.820,148.882
C09736=1189.349,38.689,-46.573,-179.484,5.820,148.881
C09737=1189.343,38.938,-46.588,-179.481,5.821,148.880
C09738=1189.338,39.188,-46.604,-179.479,5.822,148.880
C09739=1189.334,39.437,-46.619,-179.477,5.822,148.879
C09740=1189.328,39.687,-46.635,-179.473,5.824,148.878
C09741=1189.323,39.936,-46.650,-179.471,5.824,148.878
C09742=1189.318,40.186,-46.666,-179.469,5.825,148.877
C09743=1189.313,40.435,-46.681,-179.466,5.825,148.877
C09744=1189.308,40.685,-46.697,-179.464,5.826,148.876
C09745=1189.303,40.935,-46.713,-179.461,5.827,148.875
C09746=1189.299,41.184,-46.728,-179.459,5.827,148.875
C09747=1189.293,41.433,-46.743,-179.456,5.829,148.874
C09748=1189.288,41.683,-46.759,-179.453,5.830,148.874
C09749=1189.283,41.932,-46.776,-179.450,5.830,148.873
C09750=1189.279,42.181,-46.791,-179.448,5.831,148.873
C09751=1189.273,42.431,-46.806,-179.446,5.831,148.872
C09752=1189.269,42.681,-46.822,-179.443,5.832,148.871
C09753=1189.263,42.930,-46.838,-179.441,5.833,148.871
C09754=1189.258,43.180,-46.853,-179.438,5.834,148.870
C09755=1189.254,43.429,-46.869,-179.435,5.835,148.869
C09756=1189.249,43.678,-46.885,-179.433,5.836,148.869
C09757=1189.243,43.928,-46.901,-179.430,5.836,148.868
C09758=1189.239,44.178,-46.917,-179.428,5.837,148.868
C09759=1189.233,44.427,-46.932,-179.425,5.838,148.867
C09760=1189.228,44.676,-46.947,-179.422,5.839,148.867
C09761=1189.224,44.926,-46.964,-179.420,5.839,148.866
C09762=1189.219,45.175,-46.979,-179.417,5.840,148.865
C09763=1189.213,45.425,-46.995,-179.415,5.841,148.865
C09764=1189.208,45.675,-47.011,-179.412,5.841,148.864
C09765=1189.203,45.923,-47.027,-179.410,5.842,148.864
C09766=1189.199,46.172,-47.042,-179.407,5.843,148.863
C09767=1189.194,46.423,-47.058,-179.404,5.844,148.862
C09768=1189.189,46.672,-47.074,-179.402,5.845,148.862
C09769=1189.183,46.921,-47.090,-179.399,5.845,148.861
C09770=1189.179,47.171,-47.106,-179.397,5.846,148.861
C09771=1189.173,47.420,-47.122,-179.395,5.847,148.860
C09772=1189.169,47.670,-47.138,-179.391,5.848,148.859
C09773=1189.163,47.919,-47.154,-179.389,5.849,148.859
C09774=1189.159,48.168,-47.169,-179.387,5.850,148.858
C09775=1189.154,48.418,-47.186,-179.384,5.850,148.858
C09776=1189.149,48.667,-47.201,-179.381,5.851,148.857
C09777=1189.144,48.917,-47.217,-179.379,5.852,148.857
C09778=1189.139,49.166,-47.233,-179.376,5.853,148.856
C09779=1189.134,49.415,-47.249,-179.373,5.853,148.855
C09780=1189.129,49.665,-47.266,-179.371,5.854,148.855
C09781=1189.124,49.914,-47.281,-179.368,5.855,148.854
C09782=1189.119,50.164,-47.297,-179.365,5.856,148.853
C09783=1189.114,50.413,-47.313,-179.363,5.857,148.853
C09784=1189.109,50.663,-47.329,-179.360,5.857,148.852
C09785=1189.104,50.912,-47.346,-179.358,5.858,148.852
C09786=1189.099,51.162,-47.362,-179.356,5.859,148.851
C09787=1189.094,51.411,-47.378,-179.352,5.860,148.851
C09788=1189.089,51.660,-47.394,-179.350,5.861,148.850
C09789=1189.084,51.910,-47.410,-179.348,5.862,148.849
C09790=1189.079,52.159,-47.426,-179.345,5.862,148.849
C09791=1189.074,52.409,-47.442,-179.343,5.863,148.848
C09792=1189.069,52.658,-47.458,-179.340,5.864,148.848
C09793=1189.064,52.908,-47.474,-179.337,5.865,148.847
C09794=1189.059,53.157,-47.490,-179.335,5.866,148.847
C09795=1189.054,53.407,-47.506,-179.332,5.866,148.846
C09796=1189.049,53.656,-47.523,-179.330,5.867,148.845
C09797=1189.045,53.905,-47.539,-179.327,5.869,148.845
C09798=1189.039,54.155,-47.555,-179.324,5.869,148.844
C09799=1189.035,54.424,-47.572,-179.322,5.870,148.843
C09800=1189.029,54.692,-47.590,-179.319,5.871,148.843
C09801=1189.024,54.960,-47.607,-179.316,5.872,148.842
C09802=1189.019,55.229,-47.625,-179.314,5.872,148.842
C09803=1189.013,55.479,-47.641,-179.310,5.874,148.841
C09804=1189.008,55.728,-47.658,-179.308,5.875,148.841
C09805=1189.003,55.977,-47.674,-179.306,5.875,148.840
C09806=1188.999,56.227,-47.690,-179.303,5.876,148.839
C09807=1188.993,56.476,-47.707,-179.300,5.877,148.839
C09808=1188.989,56.726,-47.722,-179.298,5.878,148.838
C09809=1188.984,56.975,-47.739,-179.295,5.879,148.838
C09810=1188.979,57.224,-47.755,-179.293,5.879,148.837
C09811=1188.973,57.474,-47.772,-179.290,5.880,148.836
C09812=1188.969,57.723,-47.788,-179.287,5.882,148.836
C09813=1188.963,57.972,-47.805,-179.285,5.882,148.835
C09814=1188.959,58.222,-47.821,-179.282,5.883,148.835
C09815=1188.954,58.472,-47.837,-179.280,5.883,148.834
C09816=1188.949,58.720,-47.854,-179.277,5.885,148.833
C09817=1188.944,58.971,-47.869,-179.275,5.886,148.833
C09818=1188.939,59.220,-47.886,-179.272,5.886,148.832
C09819=1188.934,59.469,-47.903,-179.269,5.887,148.832
C09820=1188.929,59.718,-47.919,-179.267,5.888,148.831
C09821=1188.924,59.968,-47.935,-179.264,5.889,148.831
C09822=1188.920,60.218,-47.952,-179.261,5.890,148.830
C09823=1188.914,60.467,-47.969,-179.259,5.890,148.830
C09824=1188.909,60.716,-47.986,-179.256,5.892,148.829
C09825=1188.904,60.965,-48.002,-179.254,5.893,148.828
C09826=1188.900,61.215,-48.018,-179.251,5.893,148.828
C09827=1188.894,61.465,-48.035,-179.249,5.894,148.827
C09828=1188.889,61.714,-48.051,-179.246,5.895,148.827
C09829=1188.885,61.963,-48.068,-179.243,5.896,148.826
C09830=1188.880,62.212,-48.084,-179.241,5.897,148.826
C09831=1188.874,62.462,-48.102,-179.238,5.897,148.825
C09832=1188.870,62.712,-48.118,-179.235,5.899,148.824
C09833=1188.865,62.961,-48.134,-179.233,5.900,148.824
C09834=1188.860,63.210,-48.151,-179.230,5.900,148.823
C09835=1188.855,63.460,-48.168,-179.228,5.902,148.823
C09836=1188.850,63.709,-48.184,-179.225,5.902,148.822
C09837=1188.845,63.958,-48.201,-179.223,5.903,148.821
C09838=1188.840,64.208,-48.218,-179.220,5.904,148.821
C09839=1188.835,64.457,-48.234,-179.217,5.905,148.820
C09840=1188.831,64.706,-48.251,-179.215,5.906,148.820
C09841=1188.825,64.956,-48.268,-179.212,5.907,148.819
C09842=1188.820,65.205,-48.284,-179.209,5.908,148.819
C09843=1188.815,65.455,-48.301,-179.207,5.909,148.818
C09844=1188.810,65.705,-48.318,-179.204,5.909,148.817
C09845=1188.805,65.953,-48.334,-179.202,5.910,148.817
C09846=1188.801,66.203,-48.351,-179.199,5.912,148.816
C09847=1188.795,66.453,-48.368,-179.196,5.912,148.816
C09848=1188.791,66.702,-48.385,-179.194,5.913,148.815
C09849=1188.786,66.951,-48.401,-179.191,5.914,148.815
C09850=1188.781,67.201,-48.418,-179.189,5.915,148.814
C09851=1188.776,67.450,-48.435,-179.186,5.916,148.813
C09852=1188.771,67.699,-48.453,-179.184,5.917,148.813
C09853=1188.766,67.948,-48.469,-179.181,5.918,148.812
C09854=1188.762,68.198,-48.486,-179.178,5.919,148.812
C09855=1188.757,68.447,-48.503,-179.176,5.919,148.811
C09856=1188.751,68.696,-48.519,-179.173,5.921,148.811
C09857=1188.746,68.946,-48.537,-179.171,5.922,148.810
C09858=1188.742,69.196,-48.553,-179.168,5.922,148.810
C09859=1188.737,69.445,-48.571,-179.165,5.924,148.809
C09860=1188.731,69.694,-48.587,-179.163,5.925,148.808
C09861=1188.727,69.944,-48.604,-179.160,5.925,148.808
C09862=1188.722,70.193,-48.621,-179.158,5.926,148.807
C09863=1188.718,70.442,-48.638,-179.155,5.927,148.807
C09864=1188.712,70.691,-48.655,-179.153,5.928,148.806
C09865=1188.707,70.941,-48.672,-179.150,5.929,148.806
C09866=1188.702,71.191,-48.689,-179.147,5.930,148.805
C09867=1188.698,71.440,-48.706,-179.145,5.931,148.805
C09868=1188.692,71.689,-48.723,-179.142,5.932,148.804
C09869=1188.688,71.938,-48.740,-179.139,5.933,148.803
C09870=1188.682,72.188,-48.757,-179.137,5.934,148.803
C09871=1188.678,72.437,-48.774,-179.135,5.935,148.802
C09872=1188.673,72.687,-48.791,-179.131,5.936,148.802
C09873=1188.668,72.935,-48.808,-179.129,5.937,148.801
C09874=1188.663,73.185,-48.826,-179.127,5.938,148.801
C09875=1188.658,73.435,-48.842,-179.123,5.939,148.800
C09876=1188.653,73.684,-48.859,-179.121,5.940,148.800
C09877=1188.648,73.934,-48.877,-179.119,5.940,148.799
C09878=1188.644,74.183,-48.894,-179.116,5.942,148.798
C09879=1188.638,74.432,-48.911,-179.113,5.943,148.798
C09880=1188.634,74.681,-48.928,-179.111,5.943,148.797
C09881=1188.628,74.931,-48.946,-179.108,5.945,148.797
C09882=1188.624,75.180,-48.962,-179.105,5.945,148.796
C09883=1188.619,75.430,-48.980,-179.103,5.946,148.796
C09884=1188.614,75.679,-48.998,-179.100,5.948,148.795
C09885=1188.609,75.928,-49.014,-179.098,5.949,148.795
C09886=1188.604,76.177,-49.032,-179.095,5.949,148.794
C09887=1188.599,76.427,-49.049,-179.092,5.951,148.793
C09888=1188.594,76.676,-49.066,-179.090,5.951,148.793
C09889=1188.589,76.926,-49.084,-179.088,5.952,148.792
C09890=1188.585,77.175,-49.100,-179.084,5.954,148.792
C09891=1188.579,77.425,-49.118,-179.082,5.954,148.791
C09892=1188.575,77.674,-49.136,-179.080,5.955,148.791
C09893=1188.569,77.923,-49.152,-179.076,5.956,148.790
C09894=1188.565,78.172,-49.170,-179.074,5.957,148.790
C09895=1188.559,78.422,-49.187,-179.071,5.959,148.789
C09896=1188.555,78.671,-49.205,-179.069,5.960,148.788
C09897=1188.550,78.921,-49.222,-179.066,5.960,148.788
C09898=1188.545,79.170,-49.240,-179.064,5.962,148.787
C09899=1188.540,79.419,-49.257,-179.061,5.962,148.787
C09900=1188.536,79.668,-49.274,-179.059,5.963,148.786
C09901=1188.530,79.918,-49.292,-179.056,5.965,148.786
C09902=1188.525,80.167,-49.310,-179.054,5.966,148.785
C09903=1188.520,80.435,-49.327,-179.050,5.967,148.785
C09904=1188.515,80.704,-49.346,-179.048,5.967,148.784
C09905=1188.510,80.972,-49.366,-179.044,5.969,148.783
C09906=1188.504,81.241,-49.384,-179.042,5.970,148.783
C09907=1188.499,81.490,-49.402,-179.039,5.971,148.782
C09908=1188.495,81.740,-49.419,-179.037,5.972,148.782
C09909=1188.490,81.989,-49.437,-179.034,5.973,148.781
C09910=1188.485,82.239,-49.454,-179.032,5.974,148.781
C09911=1188.480,82.488,-49.472,-179.029,5.975,148.780
C09912=1188.474,82.736,-49.490,-179.026,5.977,148.780
C09913=1188.470,82.986,-49.506,-179.024,5.977,148.779
C09914=1188.465,83.235,-49.524,-179.022,5.978,148.779
C09915=1188.460,83.484,-49.542,-179.018,5.979,148.778
C09916=1188.455,83.734,-49.560,-179.016,5.980,148.777
C09917=1188.450,83.983,-49.578,-179.013,5.982,148.777
C09918=1188.446,84.232,-49.595,-179.010,5.982,148.776
C09919=1188.441,84.482,-49.612,-179.008,5.983,148.776
C09920=1188.436,84.731,-49.630,-179.005,5.984,148.775
C09921=1188.431,84.980,-49.648,-179.003,5.985,148.775
C09922=1188.426,85.230,-49.666,-179.000,5.987,148.774
C09923=1188.421,85.479,-49.683,-178.998,5.988,148.774
C09924=1188.416,85.728,-49.701,-178.995,5.988,148.773
C09925=1188.412,85.979,-49.719,-178.992,5.990,148.773
C09926=1188.407,86.228,-49.736,-178.990,5.990,148.772
C09927=1188.402,86.477,-49.754,-178.987,5.992,148.771
C09928=1188.397,86.726,-49.772,-178.984,5.993,148.771
C09929=1188.392,86.976,-49.790,-178.982,5.994,148.770
C09930=1188.387,87.225,-49.808,-178.979,5.995,148.770
C09931=1188.382,87.474,-49.826,-178.977,5.996,148.769
C09932=1188.377,87.723,-49.844,-178.974,5.997,148.769
C09933=1188.372,87.973,-49.862,-178.971,5.998,148.768
C09934=1188.367,88.222,-49.879,-178.968,6.000,148.768
C09935=1188.362,88.472,-49.897,-178.966,6.000,148.767
C09936=1188.358,88.720,-49.914,-178.963,6.001,148.767
C09937=1188.353,88.970,-49.932,-178.961,6.003,148.766
C09938=1188.348,89.219,-49.950,-178.958,6.003,148.765
C09939=1188.343,89.468,-49.968,-178.955,6.005,148.765
C09940=1188.338,89.717,-49.986,-178.953,6.006,148.764
C09941=1188.334,89.968,-50.004,-178.950,6.007,148.764
C09942=1188.329,90.217,-50.022,-178.947,6.008,148.763
C09943=1188.324,90.466,-50.040,-178.945,6.009,148.763
C09944=1188.319,90.715,-50.058,-178.943,6.011,148.762
C09945=1188.314,90.964,-50.076,-178.940,6.011,148.762
C09946=1188.309,91.214,-50.094,-178.937,6.013,148.761
C09947=1188.304,91.463,-50.112,-178.935,6.013,148.761
C09948=1188.299,91.712,-50.130,-178.932,6.015,148.760
C09949=1188.294,91.961,-50.148,-178.929,6.016,148.760
C09950=1188.290,92.211,-50.166,-178.927,6.017,148.759
C09951=1188.285,92.460,-50.184,-178.924,6.018,148.759
C09952=1188.280,92.709,-50.202,-178.922,6.019,148.758
C09953=1188.275,92.959,-50.221,-178.919,6.020,148.758
C09954=1188.270,93.208,-50.239,-178.917,6.021,148.757
C09955=1188.265,93.457,-50.256,-178.913,6.022,148.757
C09956=1188.260,93.706,-50.274,-178.911,6.023,148.756
C09957=1188.256,93.956,-50.293,-178.908,6.025,148.755
C09958=1188.251,94.205,-50.311,-178.906,6.026,148.755
C09959=1188.246,94.455,-50.329,-178.903,6.027,148.754
C09960=1188.241,94.704,-50.347,-178.901,6.028,148.754
C09961=1188.236,94.953,-50.365,-178.898,6.029,148.753
C09962=1188.232,95.203,-50.383,-178.895,6.030,148.753
C09963=1188.227,95.452,-50.401,-178.893,6.031,148.752
C09964=1188.221,95.701,-50.420,-178.890,6.033,148.752
C09965=1188.216,95.951,-50.438,-178.888,6.033,148.751
C09966=1188.212,96.199,-50.456,-178.885,6.035,148.751
C09967=1188.207,96.449,-50.475,-178.882,6.036,148.750
C09968=1188.202,96.698,-50.493,-178.879,6.037,148.750
C09969=1188.197,96.947,-50.511,-178.877,6.038,148.749
C09970=1188.192,97.197,-50.529,-178.874,6.039,148.749
C09971=1188.187,97.446,-50.547,-178.872,6.040,148.748
C09972=1188.183,97.696,-50.566,-178.869,6.042,148.748
C09973=1188.178,97.944,-50.584,-178.866,6.043,148.747
C09974=1188.173,98.194,-50.602,-178.864,6.044,148.747
C09975=1188.167,98.443,-50.621,-178.861,6.045,148.746
C09976=1188.163,98.693,-50.639,-178.858,6.047,148.746
C09977=1188.158,98.942,-50.658,-178.856,6.047,148.745
C09978=1188.154,99.191,-50.676,-178.853,6.049,148.745
C09979=1188.149,99.440,-50.694,-178.850,6.050,148.744
C09980=1188.144,99.690,-50.713,-178.848,6.051,148.744
C09981=1188.139,99.939,-50.731,-178.845,6.052,148.743
C09982=1188.134,100.188,-50.749,-178.842,6.054,148.743
C09983=1188.129,100.437,-50.767,-178.840,6.054,148.742
C09984=1188.124,100.687,-50.786,-178.837,6.056,148.742
C09985=1188.119,100.936,-50.805,-178.835,6.057,148.741
C09986=1188.115,101.185,-50.823,-178.832,6.058,148.740
C09987=1188.110,101.435,-50.841,-178.830,6.059,148.740
C09988=1188.105,101.684,-50.861,-178.826,6.060,148.739
C09989=1188.100,101.933,-50.879,-178.824,6.061,148.739
C09990=1188.095,102.182,-50.897,-178.822,6.063,148.739
C09991=1188.090,102.432,-50.916,-178.819,6.064,148.738
C09992=1188.085,102.681,-50.934,-178.816,6.065,148.738
C09993=1188.081,102.930,-50.952,-178.814,6.066,148.737
C09994=1188.076,103.180,-50.972,-178.811,6.068,148.736
C09995=1188.071,103.429,-50.990,-178.808,6.068,148.736
C09996=1188.066,103.677,-51.009,-178.806,6.070,148.735
//INST
///DATE 2021/06/15 17:24
///ATTR SC,RW,RJ
////FRAME ROBOT
///GROUP1 RB1
NOP
MOVL C00000 V=800.0 PL=0
MOVL C00001 V=800.0 PL=0
MOVL C00002 V=800.0 PL=0
MOVL C00003 V=800.0 PL=0
MOVL C00004 V=800.0 PL=0
MOVL C00005 V=800.0 PL=0
MOVL C00006 V=800.0 PL=0
MOVL C00007 V=800.0 PL=0
MOVL C00008 V=800.0 PL=0
MOVL C00009 V=800.0 PL=0
MOVL C00010 V=800.0 PL=0
MOVL C00011 V=800.0 PL=0
MOVL C00012 V=800.0 PL=0
MOVL C00013 V=800.0 PL=0
MOVL C00014 V=800.0 PL=0
MOVL C00015 V=800.0 PL=0
MOVL C00016 V=800.0 PL=0
MOVL C00017 V=800.0 PL=0
MOVL C00018 V=800.0 PL=0
MOVL C00019 V=800.0 PL=0
MOVL C00020 V=800.0 PL=0
MOVL C00021 V=800.0 PL=0
MOVL C00022 V=800.0 PL=0
MOVL C00023 V=800.0 PL=0
MOVL C00024 V=800.0 PL=0
MOVL C00025 V=800.0 PL=0
MOVL C00026 V=800.0 PL=0
MOVL C00027 V=800.0 PL=0
MOVL C00028 V=800.0 PL=0
MOVL C00029 V=800.0 PL=0
MOVL C00030 V=800.0 PL=0
MOVL C00031 V=800.0 PL=0
MOVL C00032 V=800.0 PL=0
MOVL C00033 V=800.0 PL=0
MOVL C00034 V=800.0 PL=0
MOVL C00035 V=800.0 PL=0
MOVL C00036 V=800.0 PL=0
MOVL C00037 V=800.0 PL=0
MOVL C00038 V=800.0 PL=0
MOVL C00039 V=800.0 PL=0
MOVL C00040 V=800.0 PL=0
MOVL C00041 V=800.0 PL=0
MOVL C00042 V=800.0 PL=0
MOVL C00043 V=800.0 PL=0
MOVL C00044 V=800.0 PL=0
MOVL C00045 V=800.0 PL=0
MOVL C00046 V=800.0 PL=0
MOVL C00047 V=800.0 PL=0
MOVL C00048 V=800.0 PL=0
MOVL C00049 V=800.0 PL=0
MOVL C00050 V=800.0 PL=0
MOVL C00051 V=800.0 PL=0
MOVL C00052 V=800.0 PL=0
MOVL C00053 V=800.0 PL=0
MOVL C00054 V=800.0 PL=0
MOVL C00055 V=800.0 PL=0
MOVL C00056 V=800.0 PL=0
MOVL C00057 V=800.0 PL=0
MOVL C00058 V=800.0 PL=0
MOVL C00059 V=800.0 PL=0
MOVL C00060 V=800.0 PL=0
MOVL C00061 V=800.0 PL=0
MOVL C00062 V=800.0 PL=0
MOVL C00063 V=800.0 PL=0
MOVL C00064 V=800.0 PL=0
MOVL C00065 V=800.0 PL=0
MOVL C00066 V=800.0 PL=0
MOVL C00067 V=800.0 PL=0
MOVL C00068 V=800.0 PL=0
MOVL C00069 V=800.0 PL=0
MOVL C00070 V=800.0 PL=0
MOVL C00071 V=800.0 PL=0
MOVL C00072 V=800.0 PL=0
MOVL C00073 V=800.0 PL=0
MOVL C00074 V=800.0 PL=0
MOVL C00075 V=800.0 PL=0
MOVL C00076 V=800.0 PL=0
MOVL C00077 V=800.0 PL=0
MOVL C00078 V=800.0 PL=0
MOVL C00079 V=800.0 PL=0
MOVL C00080 V=800.0 PL=0
MOVL C00081 V=800.0 PL=0
MOVL C00082 V=800.0 PL=0
MOVL C00083 V=800.0 PL=0
MOVL C00084 V=800.0 PL=0
MOVL C00085 V=800.0 PL=0
MOVL C00086 V=800.0 PL=0
MOVL C00087 V=800.0 PL=0
MOVL C00088 V=800.0 PL=0
MOVL C00089 V=800.0 PL=0
MOVL C00090 V=800.0 PL=0
MOVL C00091 V=800.0 PL=0
MOVL C00092 V=800.0 PL=0
MOVL C00093 V=800.0 PL=0
MOVL C00094 V=800.0 PL=0
MOVL C00095 V=800.0 PL=0
MOVL C00096 V=800.0 PL=0
MOVL C00097 V=800.0 PL=0
MOVL C00098 V=800.0 PL=0
MOVL C00099 V=800.0 PL=0
MOVL C00100 V=800.0 PL=0
MOVL C00101 V=800.0 PL=0
MOVL C00102 V=800.0 PL=0
MOVL C00103 V=800.0 PL=0
MOVL C00104 V=800.0 PL=0
MOVL C00105 V=800.0 PL=0
MOVL C00106 V=800.0 PL=0
MOVL C00107 V=800.0 PL=0
MOVL C00108 V=800.0 PL=0
MOVL C00109 V=800.0 PL=0
MOVL C00110 V=800.0 PL=0
MOVL C00111 V=800.0 PL=0
MOVL C00112 V=800.0 PL=0
MOVL C00113 V=800.0 PL=0
MOVL C00114 V=800.0 PL=0
MOVL C00115 V=800.0 PL=0
MOVL C00116 V=800.0 PL=0
MOVL C00117 V=800.0 PL=0
MOVL C00118 V=800.0 PL=0
MOVL C00119 V=800.0 PL=0
MOVL C00120 V=800.0 PL=0
MOVL C00121 V=800.0 PL=0
MOVL C00122 V=800.0 PL=0
MOVL C00123 V=800.0 PL=0
MOVL C00124 V=800.0 PL=0
MOVL C00125 V=800.0 PL=0
MOVL C00126 V=800.0 PL=0
MOVL C00127 V=800.0 PL=0
MOVL C00128 V=800.0 PL=0
MOVL C00129 V=800.0 PL=0
MOVL C00130 V=800.0 PL=0
MOVL C00131 V=800.0 PL=0
MOVL C00132 V=800.0 PL=0
MOVL C00133 V=800.0 PL=0
MOVL C00134 V=800.0 PL=0
MOVL C00135 V=800.0 PL=0
MOVL C00136 V=800.0 PL=0
MOVL C00137 V=800.0 PL=0
MOVL C00138 V=800.0 PL=0
MOVL C00139 V=800.0 PL=0
MOVL C00140 V=800.0 PL=0
MOVL C00141 V=800.0 PL=0
MOVL C00142 V=800.0 PL=0
MOVL C00143 V=800.0 PL=0
MOVL C00144 V=800.0 PL=0
MOVL C00145 V=800.0 PL=0
MOVL C00146 V=800.0 PL=0
MOVL C00147 V=800.0 PL=0
MOVL C00148 V=800.0 PL=0
MOVL C00149 V=800.0 PL=0
MOVL C00150 V=800.0 PL=0
MOVL C00151 V=800.0 PL=0
MOVL C00152 V=800.0 PL=0
MOVL C00153 V=800.0 PL=0
MOVL C00154 V=800.0 PL=0
MOVL C00155 V=800.0 PL=0
MOVL C00156 V=800.0 PL=0
MOVL C00157 V=800.0 PL=0
MOVL C00158 V=800.0 PL=0
MOVL C00159 V=800.0 PL=0
MOVL C00160 V=800.0 PL=0
MOVL C00161 V=800.0 PL=0
MOVL C00162 V=800.0 PL=0
MOVL C00163 V=800.0 PL=0
MOVL C00164 V=800.0 PL=0
MOVL C00165 V=800.0 PL=0
MOVL C00166 V=800.0 PL=0
MOVL C00167 V=800.0 PL=0
MOVL C00168 V=800.0 PL=0
MOVL C00169 V=800.0 PL=0
MOVL C00170 V=800.0 PL=0
MOVL C00171 V=800.0 PL=0
MOVL C00172 V=800.0 PL=0
MOVL C00173 V=800.0 PL=0
MOVL C00174 V=800.0 PL=0
MOVL C00175 V=800.0 PL=0
MOVL C00176 V=800.0 PL=0
MOVL C00177 V=800.0 PL=0
MOVL C00178 V=800.0 PL=0
MOVL C00179 V=800.0 PL=0
MOVL C00180 V=800.0 PL=0
MOVL C00181 V=800.0 PL=0
MOVL C00182 V=800.0 PL=0
MOVL C00183 V=800.0 PL=0
MOVL C00184 V=800.0 PL=0
MOVL C00185 V=800.0 PL=0
MOVL C00186 V=800.0 PL=0
MOVL C00187 V=800.0 PL=0
MOVL C00188 V=800.0 PL=0
MOVL C00189 V=800.0 PL=0
MOVL C00190 V=800.0 PL=0
MOVL C00191 V=800.0 PL=0
MOVL C00192 V=800.0 PL=0
MOVL C00193 V=800.0 PL=0
MOVL C00194 V=800.0 PL=0
MOVL C00195 V=800.0 PL=0
MOVL C00196 V=800.0 PL=0
MOVL C00197 V=800.0 PL=0
MOVL C00198 V=800.0 PL=0
MOVL C00199 V=800.0 PL=0
MOVL C00200 V=800.0 PL=0
MOVL C00201 V=800.0 PL=0
MOVL C00202 V=800.0 PL=0
MOVL C00203 V=800.0 PL=0
MOVL C00204 V=800.0 PL=0
MOVL C00205 V=800.0 PL=0
MOVL C00206 V=800.0 PL=0
MOVL C00207 V=800.0 PL=0
MOVL C00208 V=800.0 PL=0
MOVL C00209 V=800.0 PL=0
MOVL C00210 V=800.0 PL=0
MOVL C00211 V=800.0 PL=0
MOVL C00212 V=800.0 PL=0
MOVL C00213 V=800.0 PL=0
MOVL C00214 V=800.0 PL=0
MOVL C00215 V=800.0 PL=0
MOVL C00216 V=800.0 PL=0
MOVL C00217 V=800.0 PL=0
MOVL C00218 V=800.0 PL=0
MOVL C00219 V=800.0 PL=0
MOVL C00220 V=800.0 PL=0
MOVL C00221 V=800.0 PL=0
MOVL C00222 V=800.0 PL=0
MOVL C00223 V=800.0 PL=0
MOVL C00224 V=800.0 PL=0
MOVL C00225 V=800.0 PL=0
MOVL C00226 V=800.0 PL=0
MOVL C00227 V=800.0 PL=0
MOVL C00228 V=800.0 PL=0
MOVL C00229 V=800.0 PL=0
MOVL C00230 V=800.0 PL=0
MOVL C00231 V=800.0 PL=0
MOVL C00232 V=800.0 PL=0
MOVL C00233 V=800.0 PL=0
MOVL C00234 V=800.0 PL=0
MOVL C00235 V=800.0 PL=0
MOVL C00236 V=800.0 PL=0
MOVL C00237 V=800.0 PL=0
MOVL C00238 V=800.0 PL=0
MOVL C00239 V=800.0 PL=0
MOVL C00240 V=800.0 PL=0
MOVL C00241 V=800.0 PL=0
MOVL C00242 V=800.0 PL=0
MOVL C00243 V=800.0 PL=0
MOVL C00244 V=800.0 PL=0
MOVL C00245 V=800.0 PL=0
MOVL C00246 V=800.0 PL=0
MOVL C00247 V=800.0 PL=0
MOVL C00248 V=800.0 PL=0
MOVL C00249 V=800.0 PL=0
MOVL C00250 V=800.0 PL=0
MOVL C00251 V=800.0 PL=0
MOVL C00252 V=800.0 PL=0
MOVL C00253 V=800.0 PL=0
MOVL C00254 V=800.0 PL=0
MOVL C00255 V=800.0 PL=0
MOVL C00256 V=800.0 PL=0
MOVL C00257 V=800.0 PL=0
MOVL C00258 V=800.0 PL=0
MOVL C00259 V=800.0 PL=0
MOVL C00260 V=800.0 PL=0
MOVL C00261 V=800.0 PL=0
MOVL C00262 V=800.0 PL=0
MOVL C00263 V=800.0 PL=0
MOVL C00264 V=800.0 PL=0
MOVL C00265 V=800.0 PL=0
MOVL C00266 V=800.0 PL=0
MOVL C00267 V=800.0 PL=0
MOVL C00268 V=800.0 PL=0
MOVL C00269 V=800.0 PL=0
MOVL C00270 V=800.0 PL=0
MOVL C00271 V=800.0 PL=0
MOVL C00272 V=800.0 PL=0
MOVL C00273 V=800.0 PL=0
MOVL C00274 V=800.0 PL=0
MOVL C00275 V=800.0 PL=0
MOVL C00276 V=800.0 PL=0
MOVL C00277 V=800.0 PL=0
MOVL C00278 V=800.0 PL=0
MOVL C00279 V=800.0 PL=0
MOVL C00280 V=800.0 PL=0
MOVL C00281 V=800.0 PL=0
MOVL C00282 V=800.0 PL=0
MOVL C00283 V=800.0 PL=0
MOVL C00284 V=800.0 PL=0
MOVL C00285 V=800.0 PL=0
MOVL C00286 V=800.0 PL=0
MOVL C00287 V=800.0 PL=0
MOVL C00288 V=800.0 PL=0
MOVL C00289 V=800.0 PL=0
MOVL C00290 V=800.0 PL=0
MOVL C00291 V=800.0 PL=0
MOVL C00292 V=800.0 PL=0
MOVL C00293 V=800.0 PL=0
MOVL C00294 V=800.0 PL=0
MOVL C00295 V=800.0 PL=0
MOVL C00296 V=800.0 PL=0
MOVL C00297 V=800.0 PL=0
MOVL C00298 V=800.0 PL=0
MOVL C00299 V=800.0 PL=0
MOVL C00300 V=800.0 PL=0
MOVL C00301 V=800.0 PL=0
MOVL C00302 V=800.0 PL=0
MOVL C00303 V=800.0 PL=0
MOVL C00304 V=800.0 PL=0
MOVL C00305 V=800.0 PL=0
MOVL C00306 V=800.0 PL=0
MOVL C00307 V=800.0 PL=0
MOVL C00308 V=800.0 PL=0
MOVL C00309 V=800.0 PL=0
MOVL C00310 V=800.0 PL=0
MOVL C00311 V=800.0 PL=0
MOVL C00312 V=800.0 PL=0
MOVL C00313 V=800.0 PL=0
MOVL C00314 V=800.0 PL=0
MOVL C00315 V=800.0 PL=0
MOVL C00316 V=800.0 PL=0
MOVL C00317 V=800.0 PL=0
MOVL C00318 V=800.0 PL=0
MOVL C00319 V=800.0 PL=0
MOVL C00320 V=800.0 PL=0
MOVL C00321 V=800.0 PL=0
MOVL C00322 V=800.0 PL=0
MOVL C00323 V=800.0 PL=0
MOVL C00324 V=800.0 PL=0
MOVL C00325 V=800.0 PL=0
MOVL C00326 V=800.0 PL=0
MOVL C00327 V=800.0 PL=0
MOVL C00328 V=800.0 PL=0
MOVL C00329 V=800.0 PL=0
MOVL C00330 V=800.0 PL=0
MOVL C00331 V=800.0 PL=0
MOVL C00332 V=800.0 PL=0
MOVL C00333 V=800.0 PL=0
MOVL C00334 V=800.0 PL=0
MOVL C00335 V=800.0 PL=0
MOVL C00336 V=800.0 PL=0
MOVL C00337 V=800.0 PL=0
MOVL C00338 V=800.0 PL=0
MOVL C00339 V=800.0 PL=0
MOVL C00340 V=800.0 PL=0
MOVL C00341 V=800.0 PL=0
MOVL C00342 V=800.0 PL=0
MOVL C00343 V=800.0 PL=0
MOVL C00344 V=800.0 PL=0
MOVL C00345 V=800.0 PL=0
MOVL C00346 V=800.0 PL=0
MOVL C00347 V=800.0 PL=0
MOVL C00348 V=800.0 PL=0
MOVL C00349 V=800.0 PL=0
MOVL C00350 V=800.0 PL=0
MOVL C00351 V=800.0 PL=0
MOVL C00352 V=800.0 PL=0
MOVL C00353 V=800.0 PL=0
MOVL C00354 V=800.0 PL=0
MOVL C00355 V=800.0 PL=0
MOVL C00356 V=800.0 PL=0
MOVL C00357 V=800.0 PL=0
MOVL C00358 V=800.0 PL=0
MOVL C00359 V=800.0 PL=0
MOVL C00360 V=800.0 PL=0
MOVL C00361 V=800.0 PL=0
MOVL C00362 V=800.0 PL=0
MOVL C00363 V=800.0 PL=0
MOVL C00364 V=800.0 PL=0
MOVL C00365 V=800.0 PL=0
MOVL C00366 V=800.0 PL=0
MOVL C00367 V=800.0 PL=0
MOVL C00368 V=800.0 PL=0
MOVL C00369 V=800.0 PL=0
MOVL C00370 V=800.0 PL=0
MOVL C00371 V=800.0 PL=0
MOVL C00372 V=800.0 PL=0
MOVL C00373 V=800.0 PL=0
MOVL C00374 V=800.0 PL=0
MOVL C00375 V=800.0 PL=0
MOVL C00376 V=800.0 PL=0
MOVL C00377 V=800.0 PL=0
MOVL C00378 V=800.0 PL=0
MOVL C00379 V=800.0 PL=0
MOVL C00380 V=800.0 PL=0
MOVL C00381 V=800.0 PL=0
MOVL C00382 V=800.0 PL=0
MOVL C00383 V=800.0 PL=0
MOVL C00384 V=800.0 PL=0
MOVL C00385 V=800.0 PL=0
MOVL C00386 V=800.0 PL=0
MOVL C00387 V=800.0 PL=0
MOVL C00388 V=800.0 PL=0
MOVL C00389 V=800.0 PL=0
MOVL C00390 V=800.0 PL=0
MOVL C00391 V=800.0 PL=0
MOVL C00392 V=800.0 PL=0
MOVL C00393 V=800.0 PL=0
MOVL C00394 V=800.0 PL=0
MOVL C00395 V=800.0 PL=0
MOVL C00396 V=800.0 PL=0
MOVL C00397 V=800.0 PL=0
MOVL C00398 V=800.0 PL=0
MOVL C00399 V=800.0 PL=0
MOVL C00400 V=800.0 PL=0
MOVL C00401 V=800.0 PL=0
MOVL C00402 V=800.0 PL=0
MOVL C00403 V=800.0 PL=0
MOVL C00404 V=800.0 PL=0
MOVL C00405 V=800.0 PL=0
MOVL C00406 V=800.0 PL=0
MOVL C00407 V=800.0 PL=0
MOVL C00408 V=800.0 PL=0
MOVL C00409 V=800.0 PL=0
MOVL C00410 V=800.0 PL=0
MOVL C00411 V=800.0 PL=0
MOVL C00412 V=800.0 PL=0
MOVL C00413 V=800.0 PL=0
MOVL C00414 V=800.0 PL=0
MOVL C00415 V=800.0 PL=0
MOVL C00416 V=800.0 PL=0
MOVL C00417 V=800.0 PL=0
MOVL C00418 V=800.0 PL=0
MOVL C00419 V=800.0 PL=0
MOVL C00420 V=800.0 PL=0
MOVL C00421 V=800.0 PL=0
MOVL C00422 V=800.0 PL=0
MOVL C00423 V=800.0 PL=0
MOVL C00424 V=800.0 PL=0
MOVL C00425 V=800.0 PL=0
MOVL C00426 V=800.0 PL=0
MOVL C00427 V=800.0 PL=0
MOVL C00428 V=800.0 PL=0
MOVL C00429 V=800.0 PL=0
MOVL C00430 V=800.0 PL=0
MOVL C00431 V=800.0 PL=0
MOVL C00432 V=800.0 PL=0
MOVL C00433 V=800.0 PL=0
MOVL C00434 V=800.0 PL=0
MOVL C00435 V=800.0 PL=0
MOVL C00436 V=800.0 PL=0
MOVL C00437 V=800.0 PL=0
MOVL C00438 V=800.0 PL=0
MOVL C00439 V=800.0 PL=0
MOVL C00440 V=800.0 PL=0
MOVL C00441 V=800.0 PL=0
MOVL C00442 V=800.0 PL=0
MOVL C00443 V=800.0 PL=0
MOVL C00444 V=800.0 PL=0
MOVL C00445 V=800.0 PL=0
MOVL C00446 V=800.0 PL=0
MOVL C00447 V=800.0 PL=0
MOVL C00448 V=800.0 PL=0
MOVL C00449 V=800.0 PL=0
MOVL C00450 V=800.0 PL=0
MOVL C00451 V=800.0 PL=0
MOVL C00452 V=800.0 PL=0
MOVL C00453 V=800.0 PL=0
MOVL C00454 V=800.0 PL=0
MOVL C00455 V=800.0 PL=0
MOVL C00456 V=800.0 PL=0
MOVL C00457 V=800.0 PL=0
MOVL C00458 V=800.0 PL=0
MOVL C00459 V=800.0 PL=0
MOVL C00460 V=800.0 PL=0
MOVL C00461 V=800.0 PL=0
MOVL C00462 V=800.0 PL=0
MOVL C00463 V=800.0 PL=0
MOVL C00464 V=800.0 PL=0
MOVL C00465 V=800.0 PL=0
MOVL C00466 V=800.0 PL=0
MOVL C00467 V=800.0 PL=0
MOVL C00468 V=800.0 PL=0
MOVL C00469 V=800.0 PL=0
MOVL C00470 V=800.0 PL=0
MOVL C00471 V=800.0 PL=0
MOVL C00472 V=800.0 PL=0
MOVL C00473 V=800.0 PL=0
MOVL C00474 V=800.0 PL=0
MOVL C00475 V=800.0 PL=0
MOVL C00476 V=800.0 PL=0
MOVL C00477 V=800.0 PL=0
MOVL C00478 V=800.0 PL=0
MOVL C00479 V=800.0 PL=0
MOVL C00480 V=800.0 PL=0
MOVL C00481 V=800.0 PL=0
MOVL C00482 V=800.0 PL=0
MOVL C00483 V=800.0 PL=0
MOVL C00484 V=800.0 PL=0
MOVL C00485 V=800.0 PL=0
MOVL C00486 V=800.0 PL=0
MOVL C00487 V=800.0 PL=0
MOVL C00488 V=800.0 PL=0
MOVL C00489 V=800.0 PL=0
MOVL C00490 V=800.0 PL=0
MOVL C00491 V=800.0 PL=0
MOVL C00492 V=800.0 PL=0
MOVL C00493 V=800.0 PL=0
MOVL C00494 V=800.0 PL=0
MOVL C00495 V=800.0 PL=0
MOVL C00496 V=800.0 PL=0
MOVL C00497 V=800.0 PL=0
MOVL C00498 V=800.0 PL=0
MOVL C00499 V=800.0 PL=0
MOVL C00500 V=800.0 PL=0
MOVL C00501 V=800.0 PL=0
MOVL C00502 V=800.0 PL=0
MOVL C00503 V=800.0 PL=0
MOVL C00504 V=800.0 PL=0
MOVL C00505 V=800.0 PL=0
MOVL C00506 V=800.0 PL=0
MOVL C00507 V=800.0 PL=0
MOVL C00508 V=800.0 PL=0
MOVL C00509 V=800.0 PL=0
MOVL C00510 V=800.0 PL=0
MOVL C00511 V=800.0 PL=0
MOVL C00512 V=800.0 PL=0
MOVL C00513 V=800.0 PL=0
MOVL C00514 V=800.0 PL=0
MOVL C00515 V=800.0 PL=0
MOVL C00516 V=800.0 PL=0
MOVL C00517 V=800.0 PL=0
MOVL C00518 V=800.0 PL=0
MOVL C00519 V=800.0 PL=0
MOVL C00520 V=800.0 PL=0
MOVL C00521 V=800.0 PL=0
MOVL C00522 V=800.0 PL=0
MOVL C00523 V=800.0 PL=0
MOVL C00524 V=800.0 PL=0
MOVL C00525 V=800.0 PL=0
MOVL C00526 V=800.0 PL=0
MOVL C00527 V=800.0 PL=0
MOVL C00528 V=800.0 PL=0
MOVL C00529 V=800.0 PL=0
MOVL C00530 V=800.0 PL=0
MOVL C00531 V=800.0 PL=0
MOVL C00532 V=800.0 PL=0
MOVL C00533 V=800.0 PL=0
MOVL C00534 V=800.0 PL=0
MOVL C00535 V=800.0 PL=0
MOVL C00536 V=800.0 PL=0
MOVL C00537 V=800.0 PL=0
MOVL C00538 V=800.0 PL=0
MOVL C00539 V=800.0 PL=0
MOVL C00540 V=800.0 PL=0
MOVL C00541 V=800.0 PL=0
MOVL C00542 V=800.0 PL=0
MOVL C00543 V=800.0 PL=0
MOVL C00544 V=800.0 PL=0
MOVL C00545 V=800.0 PL=0
MOVL C00546 V=800.0 PL=0
MOVL C00547 V=800.0 PL=0
MOVL C00548 V=800.0 PL=0
MOVL C00549 V=800.0 PL=0
MOVL C00550 V=800.0 PL=0
MOVL C00551 V=800.0 PL=0
MOVL C00552 V=800.0 PL=0
MOVL C00553 V=800.0 PL=0
MOVL C00554 V=800.0 PL=0
MOVL C00555 V=800.0 PL=0
MOVL C00556 V=800.0 PL=0
MOVL C00557 V=800.0 PL=0
MOVL C00558 V=800.0 PL=0
MOVL C00559 V=800.0 PL=0
MOVL C00560 V=800.0 PL=0
MOVL C00561 V=800.0 PL=0
MOVL C00562 V=800.0 PL=0
MOVL C00563 V=800.0 PL=0
MOVL C00564 V=800.0 PL=0
MOVL C00565 V=800.0 PL=0
MOVL C00566 V=800.0 PL=0
MOVL C00567 V=800.0 PL=0
MOVL C00568 V=800.0 PL=0
MOVL C00569 V=800.0 PL=0
MOVL C00570 V=800.0 PL=0
MOVL C00571 V=800.0 PL=0
MOVL C00572 V=800.0 PL=0
MOVL C00573 V=800.0 PL=0
MOVL C00574 V=800.0 PL=0
MOVL C00575 V=800.0 PL=0
MOVL C00576 V=800.0 PL=0
MOVL C00577 V=800.0 PL=0
MOVL C00578 V=800.0 PL=0
MOVL C00579 V=800.0 PL=0
MOVL C00580 V=800.0 PL=0
MOVL C00581 V=800.0 PL=0
MOVL C00582 V=800.0 PL=0
MOVL C00583 V=800.0 PL=0
MOVL C00584 V=800.0 PL=0
MOVL C00585 V=800.0 PL=0
MOVL C00586 V=800.0 PL=0
MOVL C00587 V=800.0 PL=0
MOVL C00588 V=800.0 PL=0
MOVL C00589 V=800.0 PL=0
MOVL C00590 V=800.0 PL=0
MOVL C00591 V=800.0 PL=0
MOVL C00592 V=800.0 PL=0
MOVL C00593 V=800.0 PL=0
MOVL C00594 V=800.0 PL=0
MOVL C00595 V=800.0 PL=0
MOVL C00596 V=800.0 PL=0
MOVL C00597 V=800.0 PL=0
MOVL C00598 V=800.0 PL=0
MOVL C00599 V=800.0 PL=0
MOVL C00600 V=800.0 PL=0
MOVL C00601 V=800.0 PL=0
MOVL C00602 V=800.0 PL=0
MOVL C00603 V=800.0 PL=0
MOVL C00604 V=800.0 PL=0
MOVL C00605 V=800.0 PL=0
MOVL C00606 V=800.0 PL=0
MOVL C00607 V=800.0 PL=0
MOVL C00608 V=800.0 PL=0
MOVL C00609 V=800.0 PL=0
MOVL C00610 V=800.0 PL=0
MOVL C00611 V=800.0 PL=0
MOVL C00612 V=800.0 PL=0
MOVL C00613 V=800.0 PL=0
MOVL C00614 V=800.0 PL=0
MOVL C00615 V=800.0 PL=0
MOVL C00616 V=800.0 PL=0
MOVL C00617 V=800.0 PL=0
MOVL C00618 V=800.0 PL=0
MOVL C00619 V=800.0 PL=0
MOVL C00620 V=800.0 PL=0
MOVL C00621 V=800.0 PL=0
MOVL C00622 V=800.0 PL=0
MOVL C00623 V=800.0 PL=0
MOVL C00624 V=800.0 PL=0
MOVL C00625 V=800.0 PL=0
MOVL C00626 V=800.0 PL=0
MOVL C00627 V=800.0 PL=0
MOVL C00628 V=800.0 PL=0
MOVL C00629 V=800.0 PL=0
MOVL C00630 V=800.0 PL=0
MOVL C00631 V=800.0 PL=0
MOVL C00632 V=800.0 PL=0
MOVL C00633 V=800.0 PL=0
MOVL C00634 V=800.0 PL=0
MOVL C00635 V=800.0 PL=0
MOVL C00636 V=800.0 PL=0
MOVL C00637 V=800.0 PL=0
MOVL C00638 V=800.0 PL=0
MOVL C00639 V=800.0 PL=0
MOVL C00640 V=800.0 PL=0
MOVL C00641 V=800.0 PL=0
MOVL C00642 V=800.0 PL=0
MOVL C00643 V=800.0 PL=0
MOVL C00644 V=800.0 PL=0
MOVL C00645 V=800.0 PL=0
MOVL C00646 V=800.0 PL=0
MOVL C00647 V=800.0 PL=0
MOVL C00648 V=800.0 PL=0
MOVL C00649 V=800.0 PL=0
MOVL C00650 V=800.0 PL=0
MOVL C00651 V=800.0 PL=0
MOVL C00652 V=800.0 PL=0
MOVL C00653 V=800.0 PL=0
MOVL C00654 V=800.0 PL=0
MOVL C00655 V=800.0 PL=0
MOVL C00656 V=800.0 PL=0
MOVL C00657 V=800.0 PL=0
MOVL C00658 V=800.0 PL=0
MOVL C00659 V=800.0 PL=0
MOVL C00660 V=800.0 PL=0
MOVL C00661 V=800.0 PL=0
MOVL C00662 V=800.0 PL=0
MOVL C00663 V=800.0 PL=0
MOVL C00664 V=800.0 PL=0
MOVL C00665 V=800.0 PL=0
MOVL C00666 V=800.0 PL=0
MOVL C00667 V=800.0 PL=0
MOVL C00668 V=800.0 PL=0
MOVL C00669 V=800.0 PL=0
MOVL C00670 V=800.0 PL=0
MOVL C00671 V=800.0 PL=0
MOVL C00672 V=800.0 PL=0
MOVL C00673 V=800.0 PL=0
MOVL C00674 V=800.0 PL=0
MOVL C00675 V=800.0 PL=0
MOVL C00676 V=800.0 PL=0
MOVL C00677 V=800.0 PL=0
MOVL C00678 V=800.0 PL=0
MOVL C00679 V=800.0 PL=0
MOVL C00680 V=800.0 PL=0
MOVL C00681 V=800.0 PL=0
MOVL C00682 V=800.0 PL=0
MOVL C00683 V=800.0 PL=0
MOVL C00684 V=800.0 PL=0
MOVL C00685 V=800.0 PL=0
MOVL C00686 V=800.0 PL=0
MOVL C00687 V=800.0 PL=0
MOVL C00688 V=800.0 PL=0
MOVL C00689 V=800.0 PL=0
MOVL C00690 V=800.0 PL=0
MOVL C00691 V=800.0 PL=0
MOVL C00692 V=800.0 PL=0
MOVL C00693 V=800.0 PL=0
MOVL C00694 V=800.0 PL=0
MOVL C00695 V=800.0 PL=0
MOVL C00696 V=800.0 PL=0
MOVL C00697 V=800.0 PL=0
MOVL C00698 V=800.0 PL=0
MOVL C00699 V=800.0 PL=0
MOVL C00700 V=800.0 PL=0
MOVL C00701 V=800.0 PL=0
MOVL C00702 V=800.0 PL=0
MOVL C00703 V=800.0 PL=0
MOVL C00704 V=800.0 PL=0
MOVL C00705 V=800.0 PL=0
MOVL C00706 V=800.0 PL=0
MOVL C00707 V=800.0 PL=0
MOVL C00708 V=800.0 PL=0
MOVL C00709 V=800.0 PL=0
MOVL C00710 V=800.0 PL=0
MOVL C00711 V=800.0 PL=0
MOVL C00712 V=800.0 PL=0
MOVL C00713 V=800.0 PL=0
MOVL C00714 V=800.0 PL=0
MOVL C00715 V=800.0 PL=0
MOVL C00716 V=800.0 PL=0
MOVL C00717 V=800.0 PL=0
MOVL C00718 V=800.0 PL=0
MOVL C00719 V=800.0 PL=0
MOVL C00720 V=800.0 PL=0
MOVL C00721 V=800.0 PL=0
MOVL C00722 V=800.0 PL=0
MOVL C00723 V=800.0 PL=0
MOVL C00724 V=800.0 PL=0
MOVL C00725 V=800.0 PL=0
MOVL C00726 V=800.0 PL=0
MOVL C00727 V=800.0 PL=0
MOVL C00728 V=800.0 PL=0
MOVL C00729 V=800.0 PL=0
MOVL C00730 V=800.0 PL=0
MOVL C00731 V=800.0 PL=0
MOVL C00732 V=800.0 PL=0
MOVL C00733 V=800.0 PL=0
MOVL C00734 V=800.0 PL=0
MOVL C00735 V=800.0 PL=0
MOVL C00736 V=800.0 PL=0
MOVL C00737 V=800.0 PL=0
MOVL C00738 V=800.0 PL=0
MOVL C00739 V=800.0 PL=0
MOVL C00740 V=800.0 PL=0
MOVL C00741 V=800.0 PL=0
MOVL C00742 V=800.0 PL=0
MOVL C00743 V=800.0 PL=0
MOVL C00744 V=800.0 PL=0
MOVL C00745 V=800.0 PL=0
MOVL C00746 V=800.0 PL=0
MOVL C00747 V=800.0 PL=0
MOVL C00748 V=800.0 PL=0
MOVL C00749 V=800.0 PL=0
MOVL C00750 V=800.0 PL=0
MOVL C00751 V=800.0 PL=0
MOVL C00752 V=800.0 PL=0
MOVL C00753 V=800.0 PL=0
MOVL C00754 V=800.0 PL=0
MOVL C00755 V=800.0 PL=0
MOVL C00756 V=800.0 PL=0
MOVL C00757 V=800.0 PL=0
MOVL C00758 V=800.0 PL=0
MOVL C00759 V=800.0 PL=0
MOVL C00760 V=800.0 PL=0
MOVL C00761 V=800.0 PL=0
MOVL C00762 V=800.0 PL=0
MOVL C00763 V=800.0 PL=0
MOVL C00764 V=800.0 PL=0
MOVL C00765 V=800.0 PL=0
MOVL C00766 V=800.0 PL=0
MOVL C00767 V=800.0 PL=0
MOVL C00768 V=800.0 PL=0
MOVL C00769 V=800.0 PL=0
MOVL C00770 V=800.0 PL=0
MOVL C00771 V=800.0 PL=0
MOVL C00772 V=800.0 PL=0
MOVL C00773 V=800.0 PL=0
MOVL C00774 V=800.0 PL=0
MOVL C00775 V=800.0 PL=0
MOVL C00776 V=800.0 PL=0
MOVL C00777 V=800.0 PL=0
MOVL C00778 V=800.0 PL=0
MOVL C00779 V=800.0 PL=0
MOVL C00780 V=800.0 PL=0
MOVL C00781 V=800.0 PL=0
MOVL C00782 V=800.0 PL=0
MOVL C00783 V=800.0 PL=0
MOVL C00784 V=800.0 PL=0
MOVL C00785 V=800.0 PL=0
MOVL C00786 V=800.0 PL=0
MOVL C00787 V=800.0 PL=0
MOVL C00788 V=800.0 PL=0
MOVL C00789 V=800.0 PL=0
MOVL C00790 V=800.0 PL=0
MOVL C00791 V=800.0 PL=0
MOVL C00792 V=800.0 PL=0
MOVL C00793 V=800.0 PL=0
MOVL C00794 V=800.0 PL=0
MOVL C00795 V=800.0 PL=0
MOVL C00796 V=800.0 PL=0
MOVL C00797 V=800.0 PL=0
MOVL C00798 V=800.0 PL=0
MOVL C00799 V=800.0 PL=0
MOVL C00800 V=800.0 PL=0
MOVL C00801 V=800.0 PL=0
MOVL C00802 V=800.0 PL=0
MOVL C00803 V=800.0 PL=0
MOVL C00804 V=800.0 PL=0
MOVL C00805 V=800.0 PL=0
MOVL C00806 V=800.0 PL=0
MOVL C00807 V=800.0 PL=0
MOVL C00808 V=800.0 PL=0
MOVL C00809 V=800.0 PL=0
MOVL C00810 V=800.0 PL=0
MOVL C00811 V=800.0 PL=0
MOVL C00812 V=800.0 PL=0
MOVL C00813 V=800.0 PL=0
MOVL C00814 V=800.0 PL=0
MOVL C00815 V=800.0 PL=0
MOVL C00816 V=800.0 PL=0
MOVL C00817 V=800.0 PL=0
MOVL C00818 V=800.0 PL=0
MOVL C00819 V=800.0 PL=0
MOVL C00820 V=800.0 PL=0
MOVL C00821 V=800.0 PL=0
MOVL C00822 V=800.0 PL=0
MOVL C00823 V=800.0 PL=0
MOVL C00824 V=800.0 PL=0
MOVL C00825 V=800.0 PL=0
MOVL C00826 V=800.0 PL=0
MOVL C00827 V=800.0 PL=0
MOVL C00828 V=800.0 PL=0
MOVL C00829 V=800.0 PL=0
MOVL C00830 V=800.0 PL=0
MOVL C00831 V=800.0 PL=0
MOVL C00832 V=800.0 PL=0
MOVL C00833 V=800.0 PL=0
MOVL C00834 V=800.0 PL=0
MOVL C00835 V=800.0 PL=0
MOVL C00836 V=800.0 PL=0
MOVL C00837 V=800.0 PL=0
MOVL C00838 V=800.0 PL=0
MOVL C00839 V=800.0 PL=0
MOVL C00840 V=800.0 PL=0
MOVL C00841 V=800.0 PL=0
MOVL C00842 V=800.0 PL=0
MOVL C00843 V=800.0 PL=0
MOVL C00844 V=800.0 PL=0
MOVL C00845 V=800.0 PL=0
MOVL C00846 V=800.0 PL=0
MOVL C00847 V=800.0 PL=0
MOVL C00848 V=800.0 PL=0
MOVL C00849 V=800.0 PL=0
MOVL C00850 V=800.0 PL=0
MOVL C00851 V=800.0 PL=0
MOVL C00852 V=800.0 PL=0
MOVL C00853 V=800.0 PL=0
MOVL C00854 V=800.0 PL=0
MOVL C00855 V=800.0 PL=0
MOVL C00856 V=800.0 PL=0
MOVL C00857 V=800.0 PL=0
MOVL C00858 V=800.0 PL=0
MOVL C00859 V=800.0 PL=0
MOVL C00860 V=800.0 PL=0
MOVL C00861 V=800.0 PL=0
MOVL C00862 V=800.0 PL=0
MOVL C00863 V=800.0 PL=0
MOVL C00864 V=800.0 PL=0
MOVL C00865 V=800.0 PL=0
MOVL C00866 V=800.0 PL=0
MOVL C00867 V=800.0 PL=0
MOVL C00868 V=800.0 PL=0
MOVL C00869 V=800.0 PL=0
MOVL C00870 V=800.0 PL=0
MOVL C00871 V=800.0 PL=0
MOVL C00872 V=800.0 PL=0
MOVL C00873 V=800.0 PL=0
MOVL C00874 V=800.0 PL=0
MOVL C00875 V=800.0 PL=0
MOVL C00876 V=800.0 PL=0
MOVL C00877 V=800.0 PL=0
MOVL C00878 V=800.0 PL=0
MOVL C00879 V=800.0 PL=0
MOVL C00880 V=800.0 PL=0
MOVL C00881 V=800.0 PL=0
MOVL C00882 V=800.0 PL=0
MOVL C00883 V=800.0 PL=0
MOVL C00884 V=800.0 PL=0
MOVL C00885 V=800.0 PL=0
MOVL C00886 V=800.0 PL=0
MOVL C00887 V=800.0 PL=0
MOVL C00888 V=800.0 PL=0
MOVL C00889 V=800.0 PL=0
MOVL C00890 V=800.0 PL=0
MOVL C00891 V=800.0 PL=0
MOVL C00892 V=800.0 PL=0
MOVL C00893 V=800.0 PL=0
MOVL C00894 V=800.0 PL=0
MOVL C00895 V=800.0 PL=0
MOVL C00896 V=800.0 PL=0
MOVL C00897 V=800.0 PL=0
MOVL C00898 V=800.0 PL=0
MOVL C00899 V=800.0 PL=0
MOVL C00900 V=800.0 PL=0
MOVL C00901 V=800.0 PL=0
MOVL C00902 V=800.0 PL=0
MOVL C00903 V=800.0 PL=0
MOVL C00904 V=800.0 PL=0
MOVL C00905 V=800.0 PL=0
MOVL C00906 V=800.0 PL=0
MOVL C00907 V=800.0 PL=0
MOVL C00908 V=800.0 PL=0
MOVL C00909 V=800.0 PL=0
MOVL C00910 V=800.0 PL=0
MOVL C00911 V=800.0 PL=0
MOVL C00912 V=800.0 PL=0
MOVL C00913 V=800.0 PL=0
MOVL C00914 V=800.0 PL=0
MOVL C00915 V=800.0 PL=0
MOVL C00916 V=800.0 PL=0
MOVL C00917 V=800.0 PL=0
MOVL C00918 V=800.0 PL=0
MOVL C00919 V=800.0 PL=0
MOVL C00920 V=800.0 PL=0
MOVL C00921 V=800.0 PL=0
MOVL C00922 V=800.0 PL=0
MOVL C00923 V=800.0 PL=0
MOVL C00924 V=800.0 PL=0
MOVL C00925 V=800.0 PL=0
MOVL C00926 V=800.0 PL=0
MOVL C00927 V=800.0 PL=0
MOVL C00928 V=800.0 PL=0
MOVL C00929 V=800.0 PL=0
MOVL C00930 V=800.0 PL=0
MOVL C00931 V=800.0 PL=0
MOVL C00932 V=800.0 PL=0
MOVL C00933 V=800.0 PL=0
MOVL C00934 V=800.0 PL=0
MOVL C00935 V=800.0 PL=0
MOVL C00936 V=800.0 PL=0
MOVL C00937 V=800.0 PL=0
MOVL C00938 V=800.0 PL=0
MOVL C00939 V=800.0 PL=0
MOVL C00940 V=800.0 PL=0
MOVL C00941 V=800.0 PL=0
MOVL C00942 V=800.0 PL=0
MOVL C00943 V=800.0 PL=0
MOVL C00944 V=800.0 PL=0
MOVL C00945 V=800.0 PL=0
MOVL C00946 V=800.0 PL=0
MOVL C00947 V=800.0 PL=0
MOVL C00948 V=800.0 PL=0
MOVL C00949 V=800.0 PL=0
MOVL C00950 V=800.0 PL=0
MOVL C00951 V=800.0 PL=0
MOVL C00952 V=800.0 PL=0
MOVL C00953 V=800.0 PL=0
MOVL C00954 V=800.0 PL=0
MOVL C00955 V=800.0 PL=0
MOVL C00956 V=800.0 PL=0
MOVL C00957 V=800.0 PL=0
MOVL C00958 V=800.0 PL=0
MOVL C00959 V=800.0 PL=0
MOVL C00960 V=800.0 PL=0
MOVL C00961 V=800.0 PL=0
MOVL C00962 V=800.0 PL=0
MOVL C00963 V=800.0 PL=0
MOVL C00964 V=800.0 PL=0
MOVL C00965 V=800.0 PL=0
MOVL C00966 V=800.0 PL=0
MOVL C00967 V=800.0 PL=0
MOVL C00968 V=800.0 PL=0
MOVL C00969 V=800.0 PL=0
MOVL C00970 V=800.0 PL=0
MOVL C00971 V=800.0 PL=0
MOVL C00972 V=800.0 PL=0
MOVL C00973 V=800.0 PL=0
MOVL C00974 V=800.0 PL=0
MOVL C00975 V=800.0 PL=0
MOVL C00976 V=800.0 PL=0
MOVL C00977 V=800.0 PL=0
MOVL C00978 V=800.0 PL=0
MOVL C00979 V=800.0 PL=0
MOVL C00980 V=800.0 PL=0
MOVL C00981 V=800.0 PL=0
MOVL C00982 V=800.0 PL=0
MOVL C00983 V=800.0 PL=0
MOVL C00984 V=800.0 PL=0
MOVL C00985 V=800.0 PL=0
MOVL C00986 V=800.0 PL=0
MOVL C00987 V=800.0 PL=0
MOVL C00988 V=800.0 PL=0
MOVL C00989 V=800.0 PL=0
MOVL C00990 V=800.0 PL=0
MOVL C00991 V=800.0 PL=0
MOVL C00992 V=800.0 PL=0
MOVL C00993 V=800.0 PL=0
MOVL C00994 V=800.0 PL=0
MOVL C00995 V=800.0 PL=0
MOVL C00996 V=800.0 PL=0
MOVL C00997 V=800.0 PL=0
MOVL C00998 V=800.0 PL=0
MOVL C00999 V=800.0 PL=0
MOVL C01000 V=800.0 PL=0
MOVL C01001 V=800.0 PL=0
MOVL C01002 V=800.0 PL=0
MOVL C01003 V=800.0 PL=0
MOVL C01004 V=800.0 PL=0
MOVL C01005 V=800.0 PL=0
MOVL C01006 V=800.0 PL=0
MOVL C01007 V=800.0 PL=0
MOVL C01008 V=800.0 PL=0
MOVL C01009 V=800.0 PL=0
MOVL C01010 V=800.0 PL=0
MOVL C01011 V=800.0 PL=0
MOVL C01012 V=800.0 PL=0
MOVL C01013 V=800.0 PL=0
MOVL C01014 V=800.0 PL=0
MOVL C01015 V=800.0 PL=0
MOVL C01016 V=800.0 PL=0
MOVL C01017 V=800.0 PL=0
MOVL C01018 V=800.0 PL=0
MOVL C01019 V=800.0 PL=0
MOVL C01020 V=800.0 PL=0
MOVL C01021 V=800.0 PL=0
MOVL C01022 V=800.0 PL=0
MOVL C01023 V=800.0 PL=0
MOVL C01024 V=800.0 PL=0
MOVL C01025 V=800.0 PL=0
MOVL C01026 V=800.0 PL=0
MOVL C01027 V=800.0 PL=0
MOVL C01028 V=800.0 PL=0
MOVL C01029 V=800.0 PL=0
MOVL C01030 V=800.0 PL=0
MOVL C01031 V=800.0 PL=0
MOVL C01032 V=800.0 PL=0
MOVL C01033 V=800.0 PL=0
MOVL C01034 V=800.0 PL=0
MOVL C01035 V=800.0 PL=0
MOVL C01036 V=800.0 PL=0
MOVL C01037 V=800.0 PL=0
MOVL C01038 V=800.0 PL=0
MOVL C01039 V=800.0 PL=0
MOVL C01040 V=800.0 PL=0
MOVL C01041 V=800.0 PL=0
MOVL C01042 V=800.0 PL=0
MOVL C01043 V=800.0 PL=0
MOVL C01044 V=800.0 PL=0
MOVL C01045 V=800.0 PL=0
MOVL C01046 V=800.0 PL=0
MOVL C01047 V=800.0 PL=0
MOVL C01048 V=800.0 PL=0
MOVL C01049 V=800.0 PL=0
MOVL C01050 V=800.0 PL=0
MOVL C01051 V=800.0 PL=0
MOVL C01052 V=800.0 PL=0
MOVL C01053 V=800.0 PL=0
MOVL C01054 V=800.0 PL=0
MOVL C01055 V=800.0 PL=0
MOVL C01056 V=800.0 PL=0
MOVL C01057 V=800.0 PL=0
MOVL C01058 V=800.0 PL=0
MOVL C01059 V=800.0 PL=0
MOVL C01060 V=800.0 PL=0
MOVL C01061 V=800.0 PL=0
MOVL C01062 V=800.0 PL=0
MOVL C01063 V=800.0 PL=0
MOVL C01064 V=800.0 PL=0
MOVL C01065 V=800.0 PL=0
MOVL C01066 V=800.0 PL=0
MOVL C01067 V=800.0 PL=0
MOVL C01068 V=800.0 PL=0
MOVL C01069 V=800.0 PL=0
MOVL C01070 V=800.0 PL=0
MOVL C01071 V=800.0 PL=0
MOVL C01072 V=800.0 PL=0
MOVL C01073 V=800.0 PL=0
MOVL C01074 V=800.0 PL=0
MOVL C01075 V=800.0 PL=0
MOVL C01076 V=800.0 PL=0
MOVL C01077 V=800.0 PL=0
MOVL C01078 V=800.0 PL=0
MOVL C01079 V=800.0 PL=0
MOVL C01080 V=800.0 PL=0
MOVL C01081 V=800.0 PL=0
MOVL C01082 V=800.0 PL=0
MOVL C01083 V=800.0 PL=0
MOVL C01084 V=800.0 PL=0
MOVL C01085 V=800.0 PL=0
MOVL C01086 V=800.0 PL=0
MOVL C01087 V=800.0 PL=0
MOVL C01088 V=800.0 PL=0
MOVL C01089 V=800.0 PL=0
MOVL C01090 V=800.0 PL=0
MOVL C01091 V=800.0 PL=0
MOVL C01092 V=800.0 PL=0
MOVL C01093 V=800.0 PL=0
MOVL C01094 V=800.0 PL=0
MOVL C01095 V=800.0 PL=0
MOVL C01096 V=800.0 PL=0
MOVL C01097 V=800.0 PL=0
MOVL C01098 V=800.0 PL=0
MOVL C01099 V=800.0 PL=0
MOVL C01100 V=800.0 PL=0
MOVL C01101 V=800.0 PL=0
MOVL C01102 V=800.0 PL=0
MOVL C01103 V=800.0 PL=0
MOVL C01104 V=800.0 PL=0
MOVL C01105 V=800.0 PL=0
MOVL C01106 V=800.0 PL=0
MOVL C01107 V=800.0 PL=0
MOVL C01108 V=800.0 PL=0
MOVL C01109 V=800.0 PL=0
MOVL C01110 V=800.0 PL=0
MOVL C01111 V=800.0 PL=0
MOVL C01112 V=800.0 PL=0
MOVL C01113 V=800.0 PL=0
MOVL C01114 V=800.0 PL=0
MOVL C01115 V=800.0 PL=0
MOVL C01116 V=800.0 PL=0
MOVL C01117 V=800.0 PL=0
MOVL C01118 V=800.0 PL=0
MOVL C01119 V=800.0 PL=0
MOVL C01120 V=800.0 PL=0
MOVL C01121 V=800.0 PL=0
MOVL C01122 V=800.0 PL=0
MOVL C01123 V=800.0 PL=0
MOVL C01124 V=800.0 PL=0
MOVL C01125 V=800.0 PL=0
MOVL C01126 V=800.0 PL=0
MOVL C01127 V=800.0 PL=0
MOVL C01128 V=800.0 PL=0
MOVL C01129 V=800.0 PL=0
MOVL C01130 V=800.0 PL=0
MOVL C01131 V=800.0 PL=0
MOVL C01132 V=800.0 PL=0
MOVL C01133 V=800.0 PL=0
MOVL C01134 V=800.0 PL=0
MOVL C01135 V=800.0 PL=0
MOVL C01136 V=800.0 PL=0
MOVL C01137 V=800.0 PL=0
MOVL C01138 V=800.0 PL=0
MOVL C01139 V=800.0 PL=0
MOVL C01140 V=800.0 PL=0
MOVL C01141 V=800.0 PL=0
MOVL C01142 V=800.0 PL=0
MOVL C01143 V=800.0 PL=0
MOVL C01144 V=800.0 PL=0
MOVL C01145 V=800.0 PL=0
MOVL C01146 V=800.0 PL=0
MOVL C01147 V=800.0 PL=0
MOVL C01148 V=800.0 PL=0
MOVL C01149 V=800.0 PL=0
MOVL C01150 V=800.0 PL=0
MOVL C01151 V=800.0 PL=0
MOVL C01152 V=800.0 PL=0
MOVL C01153 V=800.0 PL=0
MOVL C01154 V=800.0 PL=0
MOVL C01155 V=800.0 PL=0
MOVL C01156 V=800.0 PL=0
MOVL C01157 V=800.0 PL=0
MOVL C01158 V=800.0 PL=0
MOVL C01159 V=800.0 PL=0
MOVL C01160 V=800.0 PL=0
MOVL C01161 V=800.0 PL=0
MOVL C01162 V=800.0 PL=0
MOVL C01163 V=800.0 PL=0
MOVL C01164 V=800.0 PL=0
MOVL C01165 V=800.0 PL=0
MOVL C01166 V=800.0 PL=0
MOVL C01167 V=800.0 PL=0
MOVL C01168 V=800.0 PL=0
MOVL C01169 V=800.0 PL=0
MOVL C01170 V=800.0 PL=0
MOVL C01171 V=800.0 PL=0
MOVL C01172 V=800.0 PL=0
MOVL C01173 V=800.0 PL=0
MOVL C01174 V=800.0 PL=0
MOVL C01175 V=800.0 PL=0
MOVL C01176 V=800.0 PL=0
MOVL C01177 V=800.0 PL=0
MOVL C01178 V=800.0 PL=0
MOVL C01179 V=800.0 PL=0
MOVL C01180 V=800.0 PL=0
MOVL C01181 V=800.0 PL=0
MOVL C01182 V=800.0 PL=0
MOVL C01183 V=800.0 PL=0
MOVL C01184 V=800.0 PL=0
MOVL C01185 V=800.0 PL=0
MOVL C01186 V=800.0 PL=0
MOVL C01187 V=800.0 PL=0
MOVL C01188 V=800.0 PL=0
MOVL C01189 V=800.0 PL=0
MOVL C01190 V=800.0 PL=0
MOVL C01191 V=800.0 PL=0
MOVL C01192 V=800.0 PL=0
MOVL C01193 V=800.0 PL=0
MOVL C01194 V=800.0 PL=0
MOVL C01195 V=800.0 PL=0
MOVL C01196 V=800.0 PL=0
MOVL C01197 V=800.0 PL=0
MOVL C01198 V=800.0 PL=0
MOVL C01199 V=800.0 PL=0
MOVL C01200 V=800.0 PL=0
MOVL C01201 V=800.0 PL=0
MOVL C01202 V=800.0 PL=0
MOVL C01203 V=800.0 PL=0
MOVL C01204 V=800.0 PL=0
MOVL C01205 V=800.0 PL=0
MOVL C01206 V=800.0 PL=0
MOVL C01207 V=800.0 PL=0
MOVL C01208 V=800.0 PL=0
MOVL C01209 V=800.0 PL=0
MOVL C01210 V=800.0 PL=0
MOVL C01211 V=800.0 PL=0
MOVL C01212 V=800.0 PL=0
MOVL C01213 V=800.0 PL=0
MOVL C01214 V=800.0 PL=0
MOVL C01215 V=800.0 PL=0
MOVL C01216 V=800.0 PL=0
MOVL C01217 V=800.0 PL=0
MOVL C01218 V=800.0 PL=0
MOVL C01219 V=800.0 PL=0
MOVL C01220 V=800.0 PL=0
MOVL C01221 V=800.0 PL=0
MOVL C01222 V=800.0 PL=0
MOVL C01223 V=800.0 PL=0
MOVL C01224 V=800.0 PL=0
MOVL C01225 V=800.0 PL=0
MOVL C01226 V=800.0 PL=0
MOVL C01227 V=800.0 PL=0
MOVL C01228 V=800.0 PL=0
MOVL C01229 V=800.0 PL=0
MOVL C01230 V=800.0 PL=0
MOVL C01231 V=800.0 PL=0
MOVL C01232 V=800.0 PL=0
MOVL C01233 V=800.0 PL=0
MOVL C01234 V=800.0 PL=0
MOVL C01235 V=800.0 PL=0
MOVL C01236 V=800.0 PL=0
MOVL C01237 V=800.0 PL=0
MOVL C01238 V=800.0 PL=0
MOVL C01239 V=800.0 PL=0
MOVL C01240 V=800.0 PL=0
MOVL C01241 V=800.0 PL=0
MOVL C01242 V=800.0 PL=0
MOVL C01243 V=800.0 PL=0
MOVL C01244 V=800.0 PL=0
MOVL C01245 V=800.0 PL=0
MOVL C01246 V=800.0 PL=0
MOVL C01247 V=800.0 PL=0
MOVL C01248 V=800.0 PL=0
MOVL C01249 V=800.0 PL=0
MOVL C01250 V=800.0 PL=0
MOVL C01251 V=800.0 PL=0
MOVL C01252 V=800.0 PL=0
MOVL C01253 V=800.0 PL=0
MOVL C01254 V=800.0 PL=0
MOVL C01255 V=800.0 PL=0
MOVL C01256 V=800.0 PL=0
MOVL C01257 V=800.0 PL=0
MOVL C01258 V=800.0 PL=0
MOVL C01259 V=800.0 PL=0
MOVL C01260 V=800.0 PL=0
MOVL C01261 V=800.0 PL=0
MOVL C01262 V=800.0 PL=0
MOVL C01263 V=800.0 PL=0
MOVL C01264 V=800.0 PL=0
MOVL C01265 V=800.0 PL=0
MOVL C01266 V=800.0 PL=0
MOVL C01267 V=800.0 PL=0
MOVL C01268 V=800.0 PL=0
MOVL C01269 V=800.0 PL=0
MOVL C01270 V=800.0 PL=0
MOVL C01271 V=800.0 PL=0
MOVL C01272 V=800.0 PL=0
MOVL C01273 V=800.0 PL=0
MOVL C01274 V=800.0 PL=0
MOVL C01275 V=800.0 PL=0
MOVL C01276 V=800.0 PL=0
MOVL C01277 V=800.0 PL=0
MOVL C01278 V=800.0 PL=0
MOVL C01279 V=800.0 PL=0
MOVL C01280 V=800.0 PL=0
MOVL C01281 V=800.0 PL=0
MOVL C01282 V=800.0 PL=0
MOVL C01283 V=800.0 PL=0
MOVL C01284 V=800.0 PL=0
MOVL C01285 V=800.0 PL=0
MOVL C01286 V=800.0 PL=0
MOVL C01287 V=800.0 PL=0
MOVL C01288 V=800.0 PL=0
MOVL C01289 V=800.0 PL=0
MOVL C01290 V=800.0 PL=0
MOVL C01291 V=800.0 PL=0
MOVL C01292 V=800.0 PL=0
MOVL C01293 V=800.0 PL=0
MOVL C01294 V=800.0 PL=0
MOVL C01295 V=800.0 PL=0
MOVL C01296 V=800.0 PL=0
MOVL C01297 V=800.0 PL=0
MOVL C01298 V=800.0 PL=0
MOVL C01299 V=800.0 PL=0
MOVL C01300 V=800.0 PL=0
MOVL C01301 V=800.0 PL=0
MOVL C01302 V=800.0 PL=0
MOVL C01303 V=800.0 PL=0
MOVL C01304 V=800.0 PL=0
MOVL C01305 V=800.0 PL=0
MOVL C01306 V=800.0 PL=0
MOVL C01307 V=800.0 PL=0
MOVL C01308 V=800.0 PL=0
MOVL C01309 V=800.0 PL=0
MOVL C01310 V=800.0 PL=0
MOVL C01311 V=800.0 PL=0
MOVL C01312 V=800.0 PL=0
MOVL C01313 V=800.0 PL=0
MOVL C01314 V=800.0 PL=0
MOVL C01315 V=800.0 PL=0
MOVL C01316 V=800.0 PL=0
MOVL C01317 V=800.0 PL=0
MOVL C01318 V=800.0 PL=0
MOVL C01319 V=800.0 PL=0
MOVL C01320 V=800.0 PL=0
MOVL C01321 V=800.0 PL=0
MOVL C01322 V=800.0 PL=0
MOVL C01323 V=800.0 PL=0
MOVL C01324 V=800.0 PL=0
MOVL C01325 V=800.0 PL=0
MOVL C01326 V=800.0 PL=0
MOVL C01327 V=800.0 PL=0
MOVL C01328 V=800.0 PL=0
MOVL C01329 V=800.0 PL=0
MOVL C01330 V=800.0 PL=0
MOVL C01331 V=800.0 PL=0
MOVL C01332 V=800.0 PL=0
MOVL C01333 V=800.0 PL=0
MOVL C01334 V=800.0 PL=0
MOVL C01335 V=800.0 PL=0
MOVL C01336 V=800.0 PL=0
MOVL C01337 V=800.0 PL=0
MOVL C01338 V=800.0 PL=0
MOVL C01339 V=800.0 PL=0
MOVL C01340 V=800.0 PL=0
MOVL C01341 V=800.0 PL=0
MOVL C01342 V=800.0 PL=0
MOVL C01343 V=800.0 PL=0
MOVL C01344 V=800.0 PL=0
MOVL C01345 V=800.0 PL=0
MOVL C01346 V=800.0 PL=0
MOVL C01347 V=800.0 PL=0
MOVL C01348 V=800.0 PL=0
MOVL C01349 V=800.0 PL=0
MOVL C01350 V=800.0 PL=0
MOVL C01351 V=800.0 PL=0
MOVL C01352 V=800.0 PL=0
MOVL C01353 V=800.0 PL=0
MOVL C01354 V=800.0 PL=0
MOVL C01355 V=800.0 PL=0
MOVL C01356 V=800.0 PL=0
MOVL C01357 V=800.0 PL=0
MOVL C01358 V=800.0 PL=0
MOVL C01359 V=800.0 PL=0
MOVL C01360 V=800.0 PL=0
MOVL C01361 V=800.0 PL=0
MOVL C01362 V=800.0 PL=0
MOVL C01363 V=800.0 PL=0
MOVL C01364 V=800.0 PL=0
MOVL C01365 V=800.0 PL=0
MOVL C01366 V=800.0 PL=0
MOVL C01367 V=800.0 PL=0
MOVL C01368 V=800.0 PL=0
MOVL C01369 V=800.0 PL=0
MOVL C01370 V=800.0 PL=0
MOVL C01371 V=800.0 PL=0
MOVL C01372 V=800.0 PL=0
MOVL C01373 V=800.0 PL=0
MOVL C01374 V=800.0 PL=0
MOVL C01375 V=800.0 PL=0
MOVL C01376 V=800.0 PL=0
MOVL C01377 V=800.0 PL=0
MOVL C01378 V=800.0 PL=0
MOVL C01379 V=800.0 PL=0
MOVL C01380 V=800.0 PL=0
MOVL C01381 V=800.0 PL=0
MOVL C01382 V=800.0 PL=0
MOVL C01383 V=800.0 PL=0
MOVL C01384 V=800.0 PL=0
MOVL C01385 V=800.0 PL=0
MOVL C01386 V=800.0 PL=0
MOVL C01387 V=800.0 PL=0
MOVL C01388 V=800.0 PL=0
MOVL C01389 V=800.0 PL=0
MOVL C01390 V=800.0 PL=0
MOVL C01391 V=800.0 PL=0
MOVL C01392 V=800.0 PL=0
MOVL C01393 V=800.0 PL=0
MOVL C01394 V=800.0 PL=0
MOVL C01395 V=800.0 PL=0
MOVL C01396 V=800.0 PL=0
MOVL C01397 V=800.0 PL=0
MOVL C01398 V=800.0 PL=0
MOVL C01399 V=800.0 PL=0
MOVL C01400 V=800.0 PL=0
MOVL C01401 V=800.0 PL=0
MOVL C01402 V=800.0 PL=0
MOVL C01403 V=800.0 PL=0
MOVL C01404 V=800.0 PL=0
MOVL C01405 V=800.0 PL=0
MOVL C01406 V=800.0 PL=0
MOVL C01407 V=800.0 PL=0
MOVL C01408 V=800.0 PL=0
MOVL C01409 V=800.0 PL=0
MOVL C01410 V=800.0 PL=0
MOVL C01411 V=800.0 PL=0
MOVL C01412 V=800.0 PL=0
MOVL C01413 V=800.0 PL=0
MOVL C01414 V=800.0 PL=0
MOVL C01415 V=800.0 PL=0
MOVL C01416 V=800.0 PL=0
MOVL C01417 V=800.0 PL=0
MOVL C01418 V=800.0 PL=0
MOVL C01419 V=800.0 PL=0
MOVL C01420 V=800.0 PL=0
MOVL C01421 V=800.0 PL=0
MOVL C01422 V=800.0 PL=0
MOVL C01423 V=800.0 PL=0
MOVL C01424 V=800.0 PL=0
MOVL C01425 V=800.0 PL=0
MOVL C01426 V=800.0 PL=0
MOVL C01427 V=800.0 PL=0
MOVL C01428 V=800.0 PL=0
MOVL C01429 V=800.0 PL=0
MOVL C01430 V=800.0 PL=0
MOVL C01431 V=800.0 PL=0
MOVL C01432 V=800.0 PL=0
MOVL C01433 V=800.0 PL=0
MOVL C01434 V=800.0 PL=0
MOVL C01435 V=800.0 PL=0
MOVL C01436 V=800.0 PL=0
MOVL C01437 V=800.0 PL=0
MOVL C01438 V=800.0 PL=0
MOVL C01439 V=800.0 PL=0
MOVL C01440 V=800.0 PL=0
MOVL C01441 V=800.0 PL=0
MOVL C01442 V=800.0 PL=0
MOVL C01443 V=800.0 PL=0
MOVL C01444 V=800.0 PL=0
MOVL C01445 V=800.0 PL=0
MOVL C01446 V=800.0 PL=0
MOVL C01447 V=800.0 PL=0
MOVL C01448 V=800.0 PL=0
MOVL C01449 V=800.0 PL=0
MOVL C01450 V=800.0 PL=0
MOVL C01451 V=800.0 PL=0
MOVL C01452 V=800.0 PL=0
MOVL C01453 V=800.0 PL=0
MOVL C01454 V=800.0 PL=0
MOVL C01455 V=800.0 PL=0
MOVL C01456 V=800.0 PL=0
MOVL C01457 V=800.0 PL=0
MOVL C01458 V=800.0 PL=0
MOVL C01459 V=800.0 PL=0
MOVL C01460 V=800.0 PL=0
MOVL C01461 V=800.0 PL=0
MOVL C01462 V=800.0 PL=0
MOVL C01463 V=800.0 PL=0
MOVL C01464 V=800.0 PL=0
MOVL C01465 V=800.0 PL=0
MOVL C01466 V=800.0 PL=0
MOVL C01467 V=800.0 PL=0
MOVL C01468 V=800.0 PL=0
MOVL C01469 V=800.0 PL=0
MOVL C01470 V=800.0 PL=0
MOVL C01471 V=800.0 PL=0
MOVL C01472 V=800.0 PL=0
MOVL C01473 V=800.0 PL=0
MOVL C01474 V=800.0 PL=0
MOVL C01475 V=800.0 PL=0
MOVL C01476 V=800.0 PL=0
MOVL C01477 V=800.0 PL=0
MOVL C01478 V=800.0 PL=0
MOVL C01479 V=800.0 PL=0
MOVL C01480 V=800.0 PL=0
MOVL C01481 V=800.0 PL=0
MOVL C01482 V=800.0 PL=0
MOVL C01483 V=800.0 PL=0
MOVL C01484 V=800.0 PL=0
MOVL C01485 V=800.0 PL=0
MOVL C01486 V=800.0 PL=0
MOVL C01487 V=800.0 PL=0
MOVL C01488 V=800.0 PL=0
MOVL C01489 V=800.0 PL=0
MOVL C01490 V=800.0 PL=0
MOVL C01491 V=800.0 PL=0
MOVL C01492 V=800.0 PL=0
MOVL C01493 V=800.0 PL=0
MOVL C01494 V=800.0 PL=0
MOVL C01495 V=800.0 PL=0
MOVL C01496 V=800.0 PL=0
MOVL C01497 V=800.0 PL=0
MOVL C01498 V=800.0 PL=0
MOVL C01499 V=800.0 PL=0
MOVL C01500 V=800.0 PL=0
MOVL C01501 V=800.0 PL=0
MOVL C01502 V=800.0 PL=0
MOVL C01503 V=800.0 PL=0
MOVL C01504 V=800.0 PL=0
MOVL C01505 V=800.0 PL=0
MOVL C01506 V=800.0 PL=0
MOVL C01507 V=800.0 PL=0
MOVL C01508 V=800.0 PL=0
MOVL C01509 V=800.0 PL=0
MOVL C01510 V=800.0 PL=0
MOVL C01511 V=800.0 PL=0
MOVL C01512 V=800.0 PL=0
MOVL C01513 V=800.0 PL=0
MOVL C01514 V=800.0 PL=0
MOVL C01515 V=800.0 PL=0
MOVL C01516 V=800.0 PL=0
MOVL C01517 V=800.0 PL=0
MOVL C01518 V=800.0 PL=0
MOVL C01519 V=800.0 PL=0
MOVL C01520 V=800.0 PL=0
MOVL C01521 V=800.0 PL=0
MOVL C01522 V=800.0 PL=0
MOVL C01523 V=800.0 PL=0
MOVL C01524 V=800.0 PL=0
MOVL C01525 V=800.0 PL=0
MOVL C01526 V=800.0 PL=0
MOVL C01527 V=800.0 PL=0
MOVL C01528 V=800.0 PL=0
MOVL C01529 V=800.0 PL=0
MOVL C01530 V=800.0 PL=0
MOVL C01531 V=800.0 PL=0
MOVL C01532 V=800.0 PL=0
MOVL C01533 V=800.0 PL=0
MOVL C01534 V=800.0 PL=0
MOVL C01535 V=800.0 PL=0
MOVL C01536 V=800.0 PL=0
MOVL C01537 V=800.0 PL=0
MOVL C01538 V=800.0 PL=0
MOVL C01539 V=800.0 PL=0
MOVL C01540 V=800.0 PL=0
MOVL C01541 V=800.0 PL=0
MOVL C01542 V=800.0 PL=0
MOVL C01543 V=800.0 PL=0
MOVL C01544 V=800.0 PL=0
MOVL C01545 V=800.0 PL=0
MOVL C01546 V=800.0 PL=0
MOVL C01547 V=800.0 PL=0
MOVL C01548 V=800.0 PL=0
MOVL C01549 V=800.0 PL=0
MOVL C01550 V=800.0 PL=0
MOVL C01551 V=800.0 PL=0
MOVL C01552 V=800.0 PL=0
MOVL C01553 V=800.0 PL=0
MOVL C01554 V=800.0 PL=0
MOVL C01555 V=800.0 PL=0
MOVL C01556 V=800.0 PL=0
MOVL C01557 V=800.0 PL=0
MOVL C01558 V=800.0 PL=0
MOVL C01559 V=800.0 PL=0
MOVL C01560 V=800.0 PL=0
MOVL C01561 V=800.0 PL=0
MOVL C01562 V=800.0 PL=0
MOVL C01563 V=800.0 PL=0
MOVL C01564 V=800.0 PL=0
MOVL C01565 V=800.0 PL=0
MOVL C01566 V=800.0 PL=0
MOVL C01567 V=800.0 PL=0
MOVL C01568 V=800.0 PL=0
MOVL C01569 V=800.0 PL=0
MOVL C01570 V=800.0 PL=0
MOVL C01571 V=800.0 PL=0
MOVL C01572 V=800.0 PL=0
MOVL C01573 V=800.0 PL=0
MOVL C01574 V=800.0 PL=0
MOVL C01575 V=800.0 PL=0
MOVL C01576 V=800.0 PL=0
MOVL C01577 V=800.0 PL=0
MOVL C01578 V=800.0 PL=0
MOVL C01579 V=800.0 PL=0
MOVL C01580 V=800.0 PL=0
MOVL C01581 V=800.0 PL=0
MOVL C01582 V=800.0 PL=0
MOVL C01583 V=800.0 PL=0
MOVL C01584 V=800.0 PL=0
MOVL C01585 V=800.0 PL=0
MOVL C01586 V=800.0 PL=0
MOVL C01587 V=800.0 PL=0
MOVL C01588 V=800.0 PL=0
MOVL C01589 V=800.0 PL=0
MOVL C01590 V=800.0 PL=0
MOVL C01591 V=800.0 PL=0
MOVL C01592 V=800.0 PL=0
MOVL C01593 V=800.0 PL=0
MOVL C01594 V=800.0 PL=0
MOVL C01595 V=800.0 PL=0
MOVL C01596 V=800.0 PL=0
MOVL C01597 V=800.0 PL=0
MOVL C01598 V=800.0 PL=0
MOVL C01599 V=800.0 PL=0
MOVL C01600 V=800.0 PL=0
MOVL C01601 V=800.0 PL=0
MOVL C01602 V=800.0 PL=0
MOVL C01603 V=800.0 PL=0
MOVL C01604 V=800.0 PL=0
MOVL C01605 V=800.0 PL=0
MOVL C01606 V=800.0 PL=0
MOVL C01607 V=800.0 PL=0
MOVL C01608 V=800.0 PL=0
MOVL C01609 V=800.0 PL=0
MOVL C01610 V=800.0 PL=0
MOVL C01611 V=800.0 PL=0
MOVL C01612 V=800.0 PL=0
MOVL C01613 V=800.0 PL=0
MOVL C01614 V=800.0 PL=0
MOVL C01615 V=800.0 PL=0
MOVL C01616 V=800.0 PL=0
MOVL C01617 V=800.0 PL=0
MOVL C01618 V=800.0 PL=0
MOVL C01619 V=800.0 PL=0
MOVL C01620 V=800.0 PL=0
MOVL C01621 V=800.0 PL=0
MOVL C01622 V=800.0 PL=0
MOVL C01623 V=800.0 PL=0
MOVL C01624 V=800.0 PL=0
MOVL C01625 V=800.0 PL=0
MOVL C01626 V=800.0 PL=0
MOVL C01627 V=800.0 PL=0
MOVL C01628 V=800.0 PL=0
MOVL C01629 V=800.0 PL=0
MOVL C01630 V=800.0 PL=0
MOVL C01631 V=800.0 PL=0
MOVL C01632 V=800.0 PL=0
MOVL C01633 V=800.0 PL=0
MOVL C01634 V=800.0 PL=0
MOVL C01635 V=800.0 PL=0
MOVL C01636 V=800.0 PL=0
MOVL C01637 V=800.0 PL=0
MOVL C01638 V=800.0 PL=0
MOVL C01639 V=800.0 PL=0
MOVL C01640 V=800.0 PL=0
MOVL C01641 V=800.0 PL=0
MOVL C01642 V=800.0 PL=0
MOVL C01643 V=800.0 PL=0
MOVL C01644 V=800.0 PL=0
MOVL C01645 V=800.0 PL=0
MOVL C01646 V=800.0 PL=0
MOVL C01647 V=800.0 PL=0
MOVL C01648 V=800.0 PL=0
MOVL C01649 V=800.0 PL=0
MOVL C01650 V=800.0 PL=0
MOVL C01651 V=800.0 PL=0
MOVL C01652 V=800.0 PL=0
MOVL C01653 V=800.0 PL=0
MOVL C01654 V=800.0 PL=0
MOVL C01655 V=800.0 PL=0
MOVL C01656 V=800.0 PL=0
MOVL C01657 V=800.0 PL=0
MOVL C01658 V=800.0 PL=0
MOVL C01659 V=800.0 PL=0
MOVL C01660 V=800.0 PL=0
MOVL C01661 V=800.0 PL=0
MOVL C01662 V=800.0 PL=0
MOVL C01663 V=800.0 PL=0
MOVL C01664 V=800.0 PL=0
MOVL C01665 V=800.0 PL=0
MOVL C01666 V=800.0 PL=0
MOVL C01667 V=800.0 PL=0
MOVL C01668 V=800.0 PL=0
MOVL C01669 V=800.0 PL=0
MOVL C01670 V=800.0 PL=0
MOVL C01671 V=800.0 PL=0
MOVL C01672 V=800.0 PL=0
MOVL C01673 V=800.0 PL=0
MOVL C01674 V=800.0 PL=0
MOVL C01675 V=800.0 PL=0
MOVL C01676 V=800.0 PL=0
MOVL C01677 V=800.0 PL=0
MOVL C01678 V=800.0 PL=0
MOVL C01679 V=800.0 PL=0
MOVL C01680 V=800.0 PL=0
MOVL C01681 V=800.0 PL=0
MOVL C01682 V=800.0 PL=0
MOVL C01683 V=800.0 PL=0
MOVL C01684 V=800.0 PL=0
MOVL C01685 V=800.0 PL=0
MOVL C01686 V=800.0 PL=0
MOVL C01687 V=800.0 PL=0
MOVL C01688 V=800.0 PL=0
MOVL C01689 V=800.0 PL=0
MOVL C01690 V=800.0 PL=0
MOVL C01691 V=800.0 PL=0
MOVL C01692 V=800.0 PL=0
MOVL C01693 V=800.0 PL=0
MOVL C01694 V=800.0 PL=0
MOVL C01695 V=800.0 PL=0
MOVL C01696 V=800.0 PL=0
MOVL C01697 V=800.0 PL=0
MOVL C01698 V=800.0 PL=0
MOVL C01699 V=800.0 PL=0
MOVL C01700 V=800.0 PL=0
MOVL C01701 V=800.0 PL=0
MOVL C01702 V=800.0 PL=0
MOVL C01703 V=800.0 PL=0
MOVL C01704 V=800.0 PL=0
MOVL C01705 V=800.0 PL=0
MOVL C01706 V=800.0 PL=0
MOVL C01707 V=800.0 PL=0
MOVL C01708 V=800.0 PL=0
MOVL C01709 V=800.0 PL=0
MOVL C01710 V=800.0 PL=0
MOVL C01711 V=800.0 PL=0
MOVL C01712 V=800.0 PL=0
MOVL C01713 V=800.0 PL=0
MOVL C01714 V=800.0 PL=0
MOVL C01715 V=800.0 PL=0
MOVL C01716 V=800.0 PL=0
MOVL C01717 V=800.0 PL=0
MOVL C01718 V=800.0 PL=0
MOVL C01719 V=800.0 PL=0
MOVL C01720 V=800.0 PL=0
MOVL C01721 V=800.0 PL=0
MOVL C01722 V=800.0 PL=0
MOVL C01723 V=800.0 PL=0
MOVL C01724 V=800.0 PL=0
MOVL C01725 V=800.0 PL=0
MOVL C01726 V=800.0 PL=0
MOVL C01727 V=800.0 PL=0
MOVL C01728 V=800.0 PL=0
MOVL C01729 V=800.0 PL=0
MOVL C01730 V=800.0 PL=0
MOVL C01731 V=800.0 PL=0
MOVL C01732 V=800.0 PL=0
MOVL C01733 V=800.0 PL=0
MOVL C01734 V=800.0 PL=0
MOVL C01735 V=800.0 PL=0
MOVL C01736 V=800.0 PL=0
MOVL C01737 V=800.0 PL=0
MOVL C01738 V=800.0 PL=0
MOVL C01739 V=800.0 PL=0
MOVL C01740 V=800.0 PL=0
MOVL C01741 V=800.0 PL=0
MOVL C01742 V=800.0 PL=0
MOVL C01743 V=800.0 PL=0
MOVL C01744 V=800.0 PL=0
MOVL C01745 V=800.0 PL=0
MOVL C01746 V=800.0 PL=0
MOVL C01747 V=800.0 PL=0
MOVL C01748 V=800.0 PL=0
MOVL C01749 V=800.0 PL=0
MOVL C01750 V=800.0 PL=0
MOVL C01751 V=800.0 PL=0
MOVL C01752 V=800.0 PL=0
MOVL C01753 V=800.0 PL=0
MOVL C01754 V=800.0 PL=0
MOVL C01755 V=800.0 PL=0
MOVL C01756 V=800.0 PL=0
MOVL C01757 V=800.0 PL=0
MOVL C01758 V=800.0 PL=0
MOVL C01759 V=800.0 PL=0
MOVL C01760 V=800.0 PL=0
MOVL C01761 V=800.0 PL=0
MOVL C01762 V=800.0 PL=0
MOVL C01763 V=800.0 PL=0
MOVL C01764 V=800.0 PL=0
MOVL C01765 V=800.0 PL=0
MOVL C01766 V=800.0 PL=0
MOVL C01767 V=800.0 PL=0
MOVL C01768 V=800.0 PL=0
MOVL C01769 V=800.0 PL=0
MOVL C01770 V=800.0 PL=0
MOVL C01771 V=800.0 PL=0
MOVL C01772 V=800.0 PL=0
MOVL C01773 V=800.0 PL=0
MOVL C01774 V=800.0 PL=0
MOVL C01775 V=800.0 PL=0
MOVL C01776 V=800.0 PL=0
MOVL C01777 V=800.0 PL=0
MOVL C01778 V=800.0 PL=0
MOVL C01779 V=800.0 PL=0
MOVL C01780 V=800.0 PL=0
MOVL C01781 V=800.0 PL=0
MOVL C01782 V=800.0 PL=0
MOVL C01783 V=800.0 PL=0
MOVL C01784 V=800.0 PL=0
MOVL C01785 V=800.0 PL=0
MOVL C01786 V=800.0 PL=0
MOVL C01787 V=800.0 PL=0
MOVL C01788 V=800.0 PL=0
MOVL C01789 V=800.0 PL=0
MOVL C01790 V=800.0 PL=0
MOVL C01791 V=800.0 PL=0
MOVL C01792 V=800.0 PL=0
MOVL C01793 V=800.0 PL=0
MOVL C01794 V=800.0 PL=0
MOVL C01795 V=800.0 PL=0
MOVL C01796 V=800.0 PL=0
MOVL C01797 V=800.0 PL=0
MOVL C01798 V=800.0 PL=0
MOVL C01799 V=800.0 PL=0
MOVL C01800 V=800.0 PL=0
MOVL C01801 V=800.0 PL=0
MOVL C01802 V=800.0 PL=0
MOVL C01803 V=800.0 PL=0
MOVL C01804 V=800.0 PL=0
MOVL C01805 V=800.0 PL=0
MOVL C01806 V=800.0 PL=0
MOVL C01807 V=800.0 PL=0
MOVL C01808 V=800.0 PL=0
MOVL C01809 V=800.0 PL=0
MOVL C01810 V=800.0 PL=0
MOVL C01811 V=800.0 PL=0
MOVL C01812 V=800.0 PL=0
MOVL C01813 V=800.0 PL=0
MOVL C01814 V=800.0 PL=0
MOVL C01815 V=800.0 PL=0
MOVL C01816 V=800.0 PL=0
MOVL C01817 V=800.0 PL=0
MOVL C01818 V=800.0 PL=0
MOVL C01819 V=800.0 PL=0
MOVL C01820 V=800.0 PL=0
MOVL C01821 V=800.0 PL=0
MOVL C01822 V=800.0 PL=0
MOVL C01823 V=800.0 PL=0
MOVL C01824 V=800.0 PL=0
MOVL C01825 V=800.0 PL=0
MOVL C01826 V=800.0 PL=0
MOVL C01827 V=800.0 PL=0
MOVL C01828 V=800.0 PL=0
MOVL C01829 V=800.0 PL=0
MOVL C01830 V=800.0 PL=0
MOVL C01831 V=800.0 PL=0
MOVL C01832 V=800.0 PL=0
MOVL C01833 V=800.0 PL=0
MOVL C01834 V=800.0 PL=0
MOVL C01835 V=800.0 PL=0
MOVL C01836 V=800.0 PL=0
MOVL C01837 V=800.0 PL=0
MOVL C01838 V=800.0 PL=0
MOVL C01839 V=800.0 PL=0
MOVL C01840 V=800.0 PL=0
MOVL C01841 V=800.0 PL=0
MOVL C01842 V=800.0 PL=0
MOVL C01843 V=800.0 PL=0
MOVL C01844 V=800.0 PL=0
MOVL C01845 V=800.0 PL=0
MOVL C01846 V=800.0 PL=0
MOVL C01847 V=800.0 PL=0
MOVL C01848 V=800.0 PL=0
MOVL C01849 V=800.0 PL=0
MOVL C01850 V=800.0 PL=0
MOVL C01851 V=800.0 PL=0
MOVL C01852 V=800.0 PL=0
MOVL C01853 V=800.0 PL=0
MOVL C01854 V=800.0 PL=0
MOVL C01855 V=800.0 PL=0
MOVL C01856 V=800.0 PL=0
MOVL C01857 V=800.0 PL=0
MOVL C01858 V=800.0 PL=0
MOVL C01859 V=800.0 PL=0
MOVL C01860 V=800.0 PL=0
MOVL C01861 V=800.0 PL=0
MOVL C01862 V=800.0 PL=0
MOVL C01863 V=800.0 PL=0
MOVL C01864 V=800.0 PL=0
MOVL C01865 V=800.0 PL=0
MOVL C01866 V=800.0 PL=0
MOVL C01867 V=800.0 PL=0
MOVL C01868 V=800.0 PL=0
MOVL C01869 V=800.0 PL=0
MOVL C01870 V=800.0 PL=0
MOVL C01871 V=800.0 PL=0
MOVL C01872 V=800.0 PL=0
MOVL C01873 V=800.0 PL=0
MOVL C01874 V=800.0 PL=0
MOVL C01875 V=800.0 PL=0
MOVL C01876 V=800.0 PL=0
MOVL C01877 V=800.0 PL=0
MOVL C01878 V=800.0 PL=0
MOVL C01879 V=800.0 PL=0
MOVL C01880 V=800.0 PL=0
MOVL C01881 V=800.0 PL=0
MOVL C01882 V=800.0 PL=0
MOVL C01883 V=800.0 PL=0
MOVL C01884 V=800.0 PL=0
MOVL C01885 V=800.0 PL=0
MOVL C01886 V=800.0 PL=0
MOVL C01887 V=800.0 PL=0
MOVL C01888 V=800.0 PL=0
MOVL C01889 V=800.0 PL=0
MOVL C01890 V=800.0 PL=0
MOVL C01891 V=800.0 PL=0
MOVL C01892 V=800.0 PL=0
MOVL C01893 V=800.0 PL=0
MOVL C01894 V=800.0 PL=0
MOVL C01895 V=800.0 PL=0
MOVL C01896 V=800.0 PL=0
MOVL C01897 V=800.0 PL=0
MOVL C01898 V=800.0 PL=0
MOVL C01899 V=800.0 PL=0
MOVL C01900 V=800.0 PL=0
MOVL C01901 V=800.0 PL=0
MOVL C01902 V=800.0 PL=0
MOVL C01903 V=800.0 PL=0
MOVL C01904 V=800.0 PL=0
MOVL C01905 V=800.0 PL=0
MOVL C01906 V=800.0 PL=0
MOVL C01907 V=800.0 PL=0
MOVL C01908 V=800.0 PL=0
MOVL C01909 V=800.0 PL=0
MOVL C01910 V=800.0 PL=0
MOVL C01911 V=800.0 PL=0
MOVL C01912 V=800.0 PL=0
MOVL C01913 V=800.0 PL=0
MOVL C01914 V=800.0 PL=0
MOVL C01915 V=800.0 PL=0
MOVL C01916 V=800.0 PL=0
MOVL C01917 V=800.0 PL=0
MOVL C01918 V=800.0 PL=0
MOVL C01919 V=800.0 PL=0
MOVL C01920 V=800.0 PL=0
MOVL C01921 V=800.0 PL=0
MOVL C01922 V=800.0 PL=0
MOVL C01923 V=800.0 PL=0
MOVL C01924 V=800.0 PL=0
MOVL C01925 V=800.0 PL=0
MOVL C01926 V=800.0 PL=0
MOVL C01927 V=800.0 PL=0
MOVL C01928 V=800.0 PL=0
MOVL C01929 V=800.0 PL=0
MOVL C01930 V=800.0 PL=0
MOVL C01931 V=800.0 PL=0
MOVL C01932 V=800.0 PL=0
MOVL C01933 V=800.0 PL=0
MOVL C01934 V=800.0 PL=0
MOVL C01935 V=800.0 PL=0
MOVL C01936 V=800.0 PL=0
MOVL C01937 V=800.0 PL=0
MOVL C01938 V=800.0 PL=0
MOVL C01939 V=800.0 PL=0
MOVL C01940 V=800.0 PL=0
MOVL C01941 V=800.0 PL=0
MOVL C01942 V=800.0 PL=0
MOVL C01943 V=800.0 PL=0
MOVL C01944 V=800.0 PL=0
MOVL C01945 V=800.0 PL=0
MOVL C01946 V=800.0 PL=0
MOVL C01947 V=800.0 PL=0
MOVL C01948 V=800.0 PL=0
MOVL C01949 V=800.0 PL=0
MOVL C01950 V=800.0 PL=0
MOVL C01951 V=800.0 PL=0
MOVL C01952 V=800.0 PL=0
MOVL C01953 V=800.0 PL=0
MOVL C01954 V=800.0 PL=0
MOVL C01955 V=800.0 PL=0
MOVL C01956 V=800.0 PL=0
MOVL C01957 V=800.0 PL=0
MOVL C01958 V=800.0 PL=0
MOVL C01959 V=800.0 PL=0
MOVL C01960 V=800.0 PL=0
MOVL C01961 V=800.0 PL=0
MOVL C01962 V=800.0 PL=0
MOVL C01963 V=800.0 PL=0
MOVL C01964 V=800.0 PL=0
MOVL C01965 V=800.0 PL=0
MOVL C01966 V=800.0 PL=0
MOVL C01967 V=800.0 PL=0
MOVL C01968 V=800.0 PL=0
MOVL C01969 V=800.0 PL=0
MOVL C01970 V=800.0 PL=0
MOVL C01971 V=800.0 PL=0
MOVL C01972 V=800.0 PL=0
MOVL C01973 V=800.0 PL=0
MOVL C01974 V=800.0 PL=0
MOVL C01975 V=800.0 PL=0
MOVL C01976 V=800.0 PL=0
MOVL C01977 V=800.0 PL=0
MOVL C01978 V=800.0 PL=0
MOVL C01979 V=800.0 PL=0
MOVL C01980 V=800.0 PL=0
MOVL C01981 V=800.0 PL=0
MOVL C01982 V=800.0 PL=0
MOVL C01983 V=800.0 PL=0
MOVL C01984 V=800.0 PL=0
MOVL C01985 V=800.0 PL=0
MOVL C01986 V=800.0 PL=0
MOVL C01987 V=800.0 PL=0
MOVL C01988 V=800.0 PL=0
MOVL C01989 V=800.0 PL=0
MOVL C01990 V=800.0 PL=0
MOVL C01991 V=800.0 PL=0
MOVL C01992 V=800.0 PL=0
MOVL C01993 V=800.0 PL=0
MOVL C01994 V=800.0 PL=0
MOVL C01995 V=800.0 PL=0
MOVL C01996 V=800.0 PL=0
MOVL C01997 V=800.0 PL=0
MOVL C01998 V=800.0 PL=0
MOVL C01999 V=800.0 PL=0
MOVL C02000 V=800.0 PL=0
MOVL C02001 V=800.0 PL=0
MOVL C02002 V=800.0 PL=0
MOVL C02003 V=800.0 PL=0
MOVL C02004 V=800.0 PL=0
MOVL C02005 V=800.0 PL=0
MOVL C02006 V=800.0 PL=0
MOVL C02007 V=800.0 PL=0
MOVL C02008 V=800.0 PL=0
MOVL C02009 V=800.0 PL=0
MOVL C02010 V=800.0 PL=0
MOVL C02011 V=800.0 PL=0
MOVL C02012 V=800.0 PL=0
MOVL C02013 V=800.0 PL=0
MOVL C02014 V=800.0 PL=0
MOVL C02015 V=800.0 PL=0
MOVL C02016 V=800.0 PL=0
MOVL C02017 V=800.0 PL=0
MOVL C02018 V=800.0 PL=0
MOVL C02019 V=800.0 PL=0
MOVL C02020 V=800.0 PL=0
MOVL C02021 V=800.0 PL=0
MOVL C02022 V=800.0 PL=0
MOVL C02023 V=800.0 PL=0
MOVL C02024 V=800.0 PL=0
MOVL C02025 V=800.0 PL=0
MOVL C02026 V=800.0 PL=0
MOVL C02027 V=800.0 PL=0
MOVL C02028 V=800.0 PL=0
MOVL C02029 V=800.0 PL=0
MOVL C02030 V=800.0 PL=0
MOVL C02031 V=800.0 PL=0
MOVL C02032 V=800.0 PL=0
MOVL C02033 V=800.0 PL=0
MOVL C02034 V=800.0 PL=0
MOVL C02035 V=800.0 PL=0
MOVL C02036 V=800.0 PL=0
MOVL C02037 V=800.0 PL=0
MOVL C02038 V=800.0 PL=0
MOVL C02039 V=800.0 PL=0
MOVL C02040 V=800.0 PL=0
MOVL C02041 V=800.0 PL=0
MOVL C02042 V=800.0 PL=0
MOVL C02043 V=800.0 PL=0
MOVL C02044 V=800.0 PL=0
MOVL C02045 V=800.0 PL=0
MOVL C02046 V=800.0 PL=0
MOVL C02047 V=800.0 PL=0
MOVL C02048 V=800.0 PL=0
MOVL C02049 V=800.0 PL=0
MOVL C02050 V=800.0 PL=0
MOVL C02051 V=800.0 PL=0
MOVL C02052 V=800.0 PL=0
MOVL C02053 V=800.0 PL=0
MOVL C02054 V=800.0 PL=0
MOVL C02055 V=800.0 PL=0
MOVL C02056 V=800.0 PL=0
MOVL C02057 V=800.0 PL=0
MOVL C02058 V=800.0 PL=0
MOVL C02059 V=800.0 PL=0
MOVL C02060 V=800.0 PL=0
MOVL C02061 V=800.0 PL=0
MOVL C02062 V=800.0 PL=0
MOVL C02063 V=800.0 PL=0
MOVL C02064 V=800.0 PL=0
MOVL C02065 V=800.0 PL=0
MOVL C02066 V=800.0 PL=0
MOVL C02067 V=800.0 PL=0
MOVL C02068 V=800.0 PL=0
MOVL C02069 V=800.0 PL=0
MOVL C02070 V=800.0 PL=0
MOVL C02071 V=800.0 PL=0
MOVL C02072 V=800.0 PL=0
MOVL C02073 V=800.0 PL=0
MOVL C02074 V=800.0 PL=0
MOVL C02075 V=800.0 PL=0
MOVL C02076 V=800.0 PL=0
MOVL C02077 V=800.0 PL=0
MOVL C02078 V=800.0 PL=0
MOVL C02079 V=800.0 PL=0
MOVL C02080 V=800.0 PL=0
MOVL C02081 V=800.0 PL=0
MOVL C02082 V=800.0 PL=0
MOVL C02083 V=800.0 PL=0
MOVL C02084 V=800.0 PL=0
MOVL C02085 V=800.0 PL=0
MOVL C02086 V=800.0 PL=0
MOVL C02087 V=800.0 PL=0
MOVL C02088 V=800.0 PL=0
MOVL C02089 V=800.0 PL=0
MOVL C02090 V=800.0 PL=0
MOVL C02091 V=800.0 PL=0
MOVL C02092 V=800.0 PL=0
MOVL C02093 V=800.0 PL=0
MOVL C02094 V=800.0 PL=0
MOVL C02095 V=800.0 PL=0
MOVL C02096 V=800.0 PL=0
MOVL C02097 V=800.0 PL=0
MOVL C02098 V=800.0 PL=0
MOVL C02099 V=800.0 PL=0
MOVL C02100 V=800.0 PL=0
MOVL C02101 V=800.0 PL=0
MOVL C02102 V=800.0 PL=0
MOVL C02103 V=800.0 PL=0
MOVL C02104 V=800.0 PL=0
MOVL C02105 V=800.0 PL=0
MOVL C02106 V=800.0 PL=0
MOVL C02107 V=800.0 PL=0
MOVL C02108 V=800.0 PL=0
MOVL C02109 V=800.0 PL=0
MOVL C02110 V=800.0 PL=0
MOVL C02111 V=800.0 PL=0
MOVL C02112 V=800.0 PL=0
MOVL C02113 V=800.0 PL=0
MOVL C02114 V=800.0 PL=0
MOVL C02115 V=800.0 PL=0
MOVL C02116 V=800.0 PL=0
MOVL C02117 V=800.0 PL=0
MOVL C02118 V=800.0 PL=0
MOVL C02119 V=800.0 PL=0
MOVL C02120 V=800.0 PL=0
MOVL C02121 V=800.0 PL=0
MOVL C02122 V=800.0 PL=0
MOVL C02123 V=800.0 PL=0
MOVL C02124 V=800.0 PL=0
MOVL C02125 V=800.0 PL=0
MOVL C02126 V=800.0 PL=0
MOVL C02127 V=800.0 PL=0
MOVL C02128 V=800.0 PL=0
MOVL C02129 V=800.0 PL=0
MOVL C02130 V=800.0 PL=0
MOVL C02131 V=800.0 PL=0
MOVL C02132 V=800.0 PL=0
MOVL C02133 V=800.0 PL=0
MOVL C02134 V=800.0 PL=0
MOVL C02135 V=800.0 PL=0
MOVL C02136 V=800.0 PL=0
MOVL C02137 V=800.0 PL=0
MOVL C02138 V=800.0 PL=0
MOVL C02139 V=800.0 PL=0
MOVL C02140 V=800.0 PL=0
MOVL C02141 V=800.0 PL=0
MOVL C02142 V=800.0 PL=0
MOVL C02143 V=800.0 PL=0
MOVL C02144 V=800.0 PL=0
MOVL C02145 V=800.0 PL=0
MOVL C02146 V=800.0 PL=0
MOVL C02147 V=800.0 PL=0
MOVL C02148 V=800.0 PL=0
MOVL C02149 V=800.0 PL=0
MOVL C02150 V=800.0 PL=0
MOVL C02151 V=800.0 PL=0
MOVL C02152 V=800.0 PL=0
MOVL C02153 V=800.0 PL=0
MOVL C02154 V=800.0 PL=0
